KUKA KRL program: MyProgram_034().src

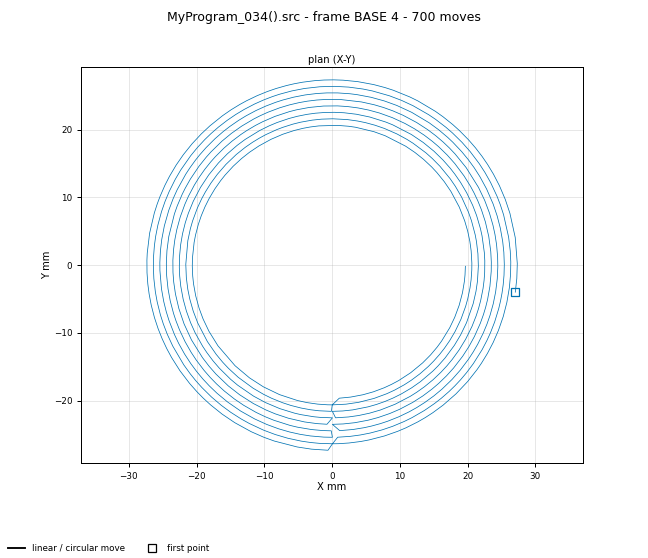
[picture p0: tool path of MyProgram_034().src in frame BASE 4, 700 of 700 moves have a stored position in this frame; points joined in program order, loops and branches not executed]
&ACCESS RVP
&REL 1
&PARAM TEMPLATE = C:\KRC\Roboter\Template\vorgabe
&PARAM EDITMASK = *
DEF MyProgram_034()
; ---- Setting reference (Base) ----
$BASE = BASE_DATA[4]

; --------------------------
; ---- Setting tool (TCP) ----
$TOOL = TOOL_DATA[3]
; --------------------------

$VEL.CP = VEL_APROX_PRINT
Startdeposition()
$VEL.CP = VEL_PRINT
LIN {X 27.0548,Y -4.0022,Z 60,A -14.7192,B 24.8252,C -3.0498,E1 25.1584,E2 -622.5769} C_DIS
LIN {X 27.276,Y -1.9895,Z 60,A -9.9625,B 24.8229,C -3.0695,E1 25.1596,E2 -627.352} C_DIS
LIN {X 27.3471,Y 0.2163,Z 60,A -4.9436,B 24.8206,C -3.0888,E1 25.1596,E2 -632.3869} C_DIS
LIN {X 27.0427,Y 4.0823,Z 60,A 3.1933,B 24.8177,C -3.1139,E1 25.1571,E2 -640.5351} C_DIS
LIN {X 26.2619,Y 7.6301,Z 60,A 9.5753,B 24.8168,C -3.1215,E1 25.1528,E2 -646.8981} C_DIS
LIN {X 25.5723,Y 9.6957,Z 60,A 14.6425,B 24.8145,C -3.1407,E1 25.1481,E2 -651.9824} C_DIS
LIN {X 24.7146,Y 11.7115,Z 60,A 18.9352,B 24.8135,C -3.1497,E1 25.1432,E2 -656.2733} C_DIS
LIN {X 23.8276,Y 13.424,Z 60,A 22.7576,B 24.8125,C -3.1579,E1 25.1381,E2 -660.0948} C_DIS
LIN {X 22.9582,Y 14.8622,Z 60,A 26.1439,B 24.8116,C -3.1652,E1 25.1331,E2 -663.4815} C_DIS
LIN {X 22.1384,Y 16.0578,Z 60,A 28.9814,B 24.811,C -3.1703,E1 25.1285,E2 -666.3172} C_DIS
LIN {X 21.1745,Y 17.3093,Z 60,A 32.8226,B 24.8093,C -3.1841,E1 25.1218,E2 -670.1731} C_DIS
LIN {X 20.1397,Y 18.5025,Z 60,A 35.9451,B 24.8087,C -3.1892,E1 25.116,E2 -673.2939} C_DIS
LIN {X 18.8106,Y 19.8529,Z 60,A 39.9521,B 24.8077,C -3.1977,E1 25.108,E2 -677.3042} C_DIS
LIN {X 17.8285,Y 20.7391,Z 60,A 42.6684,B 24.8071,C -3.2024,E1 25.1023,E2 -680.0209} C_DIS
LIN {X 16.3808,Y 21.9002,Z 60,A 46.4204,B 24.8065,C -3.2077,E1 25.094,E2 -683.7718} C_DIS
LIN {X 15.2507,Y 22.7016,Z 60,A 50.0968,B 24.8049,C -3.2207,E1 25.0855,E2 -687.4666} C_DIS
LIN {X 12.664,Y 24.2399,Z 60,A 55.4757,B 24.8051,C -3.2195,E1 25.0725,E2 -692.8267} C_DIS
LIN {X 11.4734,Y 24.8254,Z 60,A 58.7236,B 24.8041,C -3.2275,E1 25.0642,E2 -696.0853} C_DIS
LIN {X 9.042,Y 25.8106,Z 60,A 63.8728,B 24.8039,C -3.2292,E1 25.0508,E2 -701.2272} C_DIS
LIN {X 7.8177,Y 26.2072,Z 60,A 66.6148,B 24.8036,C -3.2316,E1 25.0435,E2 -703.97} C_DIS
LIN {X 6.141,Y 26.6504,Z 60,A 70.1776,B 24.8034,C -3.2329,E1 25.0339,E2 -707.5308} C_DIS
LIN {X 3.7878,Y 27.0854,Z 60,A 75.9719,B 24.8023,C -3.2419,E1 25.0179,E2 -713.3405} C_DIS
LIN {X 1.6343,Y 27.2996,Z 60,A 79.5933,B 24.8033,C -3.2337,E1 25.0078,E2 -716.9407} C_DIS
LIN {X 0.2341,Y 27.348,Z 60,A 82.5895,B 24.8033,C -3.2339,E1 24.9995,E2 -719.9368} C_DIS
LIN {X -1.1756,Y 27.3235,Z 60,A 85.9478,B 24.803,C -3.2366,E1 24.9901,E2 -723.3021} C_DIS
LIN {X -2.5854,Y 27.2262,Z 60,A 88.7053,B 24.8034,C -3.2334,E1 24.9824,E2 -726.0534} C_DIS
LIN {X -4.3352,Y 27.003,Z 60,A 92.0727,B 24.804,C -3.2283,E1 24.9731,E2 -729.4114} C_DIS
LIN {X -5.5747,Y 26.7748,Z 60,A 94.7372,B 24.8042,C -3.2265,E1 24.9658,E2 -732.0744} C_DIS
LIN {X -6.7187,Y 26.5103,Z 60,A 97.2104,B 24.8045,C -3.2243,E1 24.9591,E2 -734.5458} C_DIS
LIN {X -8.2695,Y 26.0682,Z 60,A 100.3423,B 24.8051,C -3.2187,E1 24.9508,E2 -737.6697} C_DIS
LIN {X -9.553,Y 25.6257,Z 60,A 103.726,B 24.8051,C -3.2195,E1 24.9419,E2 -741.0618} C_DIS
LIN {X -11.0562,Y 25.0141,Z 60,A 107.0784,B 24.8057,C -3.2144,E1 24.9333,E2 -744.4097} C_DIS
LIN {X -12.6311,Y 24.2572,Z 60,A 110.2156,B 24.8068,C -3.2047,E1 24.9254,E2 -747.5321} C_DIS
LIN {X -13.6382,Y 23.7057,Z 60,A 112.807,B 24.8072,C -3.2021,E1 24.9191,E2 -750.1246} C_DIS
LIN {X -14.9175,Y 22.9225,Z 60,A 116.3286,B 24.8075,C -3.1991,E1 24.9108,E2 -753.6502} C_DIS
LIN {X -16.1878,Y 22.0436,Z 60,A 119.8069,B 24.8081,C -3.1944,E1 24.9029,E2 -757.1295} C_DIS
LIN {X -18.0508,Y 20.546,Z 60,A 124.7797,B 24.8094,C -3.1834,E1 24.8923,E2 -762.0951} C_DIS
LIN {X -19.3253,Y 19.3515,Z 60,A 128.3639,B 24.8105,C -3.1744,E1 24.8851,E2 -765.6727} C_DIS
LIN {X -20.6728,Y 17.905,Z 60,A 133.0331,B 24.8113,C -3.1678,E1 24.8764,E2 -770.347} C_DIS
LIN {X -21.9574,Y 16.304,Z 60,A 136.9144,B 24.813,C -3.1539,E1 24.8698,E2 -774.2135} C_DIS
LIN {X -23.0224,Y 14.7624,Z 60,A 140.9378,B 24.8141,C -3.1439,E1 24.8636,E2 -778.2331} C_DIS
LIN {X -24.0135,Y 13.0887,Z 60,A 144.7588,B 24.8157,C -3.1309,E1 24.8583,E2 -782.0428} C_DIS
LIN {X -24.6915,Y 11.7597,Z 60,A 148.0146,B 24.8167,C -3.1227,E1 24.8543,E2 -785.2965} C_DIS
LIN {X -25.4087,Y 10.1165,Z 60,A 151.5582,B 24.8181,C -3.1103,E1 24.8505,E2 -788.8302} C_DIS
LIN {X -25.8191,Y 9.0175,Z 60,A 154.1643,B 24.8189,C -3.1038,E1 24.8481,E2 -791.4355} C_DIS
LIN {X -26.2429,Y 7.6978,Z 60,A 157.7395,B 24.8194,C -3.0991,E1 24.8452,E2 -795.02} C_DIS
LIN {X -26.9423,Y 4.7003,Z 60,A 164.4262,B 24.8216,C -3.0806,E1 24.8414,E2 -801.7017} C_DIS
LIN {X -27.2903,Y 1.7841,Z 60,A 169.5574,B 24.8245,C -3.0552,E1 24.84,E2 -806.8029} C_DIS
LIN {X -27.3397,Y 0.7102,Z 60,A 172.2916,B 24.825,C -3.0511,E1 24.8398,E2 -809.5437} C_DIS
LIN {X -27.3254,Y -1.1279,Z 60,A 176.1128,B 24.8264,C -3.0389,E1 24.84,E2 -813.3588} C_DIS
LIN {X -27.2072,Y -2.7805,Z 60,A 179.4041,B 24.8278,C -3.0271,E1 24.8408,E2 -816.6416} C_DIS
LIN {X -27.0158,Y -4.2561,Z 60,A -177.359,B 24.8288,C -3.0183,E1 24.8421,E2 -819.8767} C_DIS
LIN {X -26.7044,Y -5.9026,Z 60,A -173.7332,B 24.8299,C -3.0085,E1 24.8442,E2 -823.5003} C_DIS
LIN {X -26.2251,Y -7.7583,Z 60,A -169.3981,B 24.831,C -2.9986,E1 24.8474,E2 -827.837} C_DIS
LIN {X -25.681,Y -9.4042,Z 60,A -166.0791,B 24.8324,C -2.9862,E1 24.8505,E2 -831.1452} C_DIS
LIN {X -25.091,Y -10.8804,Z 60,A -163.0196,B 24.8336,C -2.9752,E1 24.8538,E2 -834.1952} C_DIS
LIN {X -24.4098,Y -12.3345,Z 60,A -159.3572,B 24.8344,C -2.968,E1 24.8582,E2 -837.8602} C_DIS
LIN {X -23.7002,Y -13.6473,Z 60,A -156.0691,B 24.8352,C -2.9609,E1 24.8627,E2 -841.1485} C_DIS
LIN {X -22.4555,Y -15.6113,Z 60,A -150.8,B 24.8363,C -2.9515,E1 24.8709,E2 -846.4215} C_DIS
LIN {X -21.0274,Y -17.4874,Z 60,A -146.2708,B 24.8379,C -2.9373,E1 24.8787,E2 -850.938} C_DIS
LIN {X -19.9376,Y -18.7205,Z 60,A -143.0013,B 24.8388,C -2.9286,E1 24.8848,E2 -854.2012} C_DIS
LIN {X -19.0275,Y -19.6448,Z 60,A -140.3601,B 24.8395,C -2.9225,E1 24.8901,E2 -856.839} C_DIS
LIN {X -17.962,Y -20.6236,Z 60,A -137.0049,B 24.8399,C -2.9191,E1 24.8971,E2 -860.1993} C_DIS
LIN {X -16.2373,Y -22.0074,Z 60,A -131.962,B 24.8404,C -2.9142,E1 24.9083,E2 -865.2488} C_DIS
LIN {X -14.3669,Y -23.2712,Z 60,A -127.2621,B 24.8412,C -2.9069,E1 24.9193,E2 -869.9464} C_DIS
LIN {X -11.9291,Y -24.6102,Z 60,A -121.5891,B 24.8422,C -2.8984,E1 24.9333,E2 -875.6147} C_DIS
LIN {X -10.075,Y -25.4254,Z 60,A -117.4657,B 24.8427,C -2.8932,E1 24.9439,E2 -879.735} C_DIS
LIN {X -8.5417,Y -25.9801,Z 60,A -113.2565,B 24.8423,C -2.8973,E1 24.9551,E2 -883.9619} C_DIS
LIN {X -5.1473,Y -26.86,Z 60,A -107.1176,B 24.8438,C -2.883,E1 24.9717,E2 -890.075} C_DIS
LIN {X -3.0426,Y -27.1795,Z 60,A -101.5966,B 24.8429,C -2.8918,E1 24.9871,E2 -895.6211} C_DIS
LIN {X -0.6027,Y -27.3425,Z 60,A -97.5116,B 24.8439,C -2.8825,E1 24.9984,E2 -899.6849} C_DIS
LIN {X -0.6027,Y -27.3425,Z 60,A -97.5116,B 24.8439,C -2.8825,E1 24.9984,E2 -899.6849} C_DIS
Enddeposition()
LIN {X 0.0589,Y -26.3872,Z 60,A -97.338,B 24.8433,C -2.8883,E1 24.9989,E2 -899.8724} C_DIS
Startdeposition()
$VEL.CP = VEL_PRINT
LIN {X -1.8545,Y -26.3253,Z 60,A -101.7289,B 24.8435,C -2.8859,E1 24.9867,E2 -895.4746} C_DIS
LIN {X -3.1824,Y -26.198,Z 60,A -104.3677,B 24.8432,C -2.8884,E1 24.9794,E2 -892.8403} C_DIS
LIN {X -4.5794,Y -25.9906,Z 60,A -107.6972,B 24.8434,C -2.887,E1 24.9702,E2 -889.5044} C_DIS
LIN {X -6.5439,Y -25.5663,Z 60,A -112.5834,B 24.8436,C -2.8849,E1 24.9569,E2 -884.6068} C_DIS
LIN {X -8.376,Y -25.0259,Z 60,A -116.0454,B 24.8427,C -2.8933,E1 24.9477,E2 -881.1587} C_DIS
LIN {X -10.101,Y -24.3809,Z 60,A -120.796,B 24.8429,C -2.8913,E1 24.9353,E2 -876.3929} C_DIS
LIN {X -12.22,Y -23.3909,Z 60,A -125.0898,B 24.8416,C -2.9031,E1 24.9246,E2 -872.116} C_DIS
LIN {X -13.4081,Y -22.731,Z 60,A -128.3851,B 24.8415,C -2.9046,E1 24.9166,E2 -868.8145} C_DIS
LIN {X -14.9597,Y -21.7411,Z 60,A -131.9408,B 24.8405,C -2.9138,E1 24.9083,E2 -865.2692} C_DIS
LIN {X -16.352,Y -20.7143,Z 60,A -136.4907,B 24.8404,C -2.9147,E1 24.8982,E2 -860.7052} C_DIS
LIN {X -17.8054,Y -19.4789,Z 60,A -140.2956,B 24.8392,C -2.9249,E1 24.8902,E2 -856.9093} C_DIS
LIN {X -19.2341,Y -18.0698,Z 60,A -144.562,B 24.8382,C -2.9344,E1 24.8819,E2 -852.6477} C_DIS
LIN {X -20.1352,Y -17.0603,Z 60,A -147.365,B 24.8374,C -2.9418,E1 24.8767,E2 -849.8496} C_DIS
LIN {X -20.9498,Y -16.0494,Z 60,A -150.3147,B 24.8367,C -2.9475,E1 24.8717,E2 -846.8996} C_DIS
LIN {X -21.8937,Y -14.7357,Z 60,A -154.7545,B 24.8364,C -2.9504,E1 24.8646,E2 -842.4449} C_DIS
LIN {X -23.5206,Y -11.969,Z 60,A -160.9111,B 24.8338,C -2.9735,E1 24.8563,E2 -836.3111} C_DIS
LIN {X -24.3328,Y -10.2164,Z 60,A -165.4742,B 24.8328,C -2.9829,E1 24.8511,E2 -831.7455} C_DIS
LIN {X -24.9188,Y -8.6894,Z 60,A -168.4952,B 24.8313,C -2.9961,E1 24.8482,E2 -828.739} C_DIS
LIN {X -25.3556,Y -7.3183,Z 60,A -171.8754,B 24.8304,C -3.0038,E1 24.8455,E2 -825.3577} C_DIS
LIN {X -25.8217,Y -5.4498,Z 60,A -176.6121,B 24.8293,C -3.0132,E1 24.8425,E2 -820.6158} C_DIS
LIN {X -26.0936,Y -3.9506,Z 60,A -179.4841,B 24.8279,C -3.0256,E1 24.8412,E2 -817.7565} C_DIS
LIN {X -26.3148,Y -1.9967,Z 60,A 176.035,B 24.8266,C -3.0376,E1 24.84,E2 -813.2775} C_DIS
LIN {X -26.3891,Y -0.2353,Z 60,A 172.4842,B 24.825,C -3.051,E1 24.8398,E2 -809.7374} C_DIS
LIN {X -26.3608,Y 1.251,Z 60,A 169.2644,B 24.8238,C -3.0611,E1 24.8401,E2 -806.5224} C_DIS
LIN {X -26.2322,Y 2.8893,Z 60,A 165.3007,B 24.8228,C -3.0701,E1 24.8411,E2 -802.5565} C_DIS
LIN {X -26.0485,Y 4.2383,Z 60,A 162.277,B 24.8218,C -3.079,E1 24.8424,E2 -799.5359} C_DIS
LIN {X -25.721,Y 5.9053,Z 60,A 158.6703,B 24.8204,C -3.0908,E1 24.8445,E2 -795.9363} C_DIS
LIN {X -25.1844,Y 7.8876,Z 60,A 154.2854,B 24.8188,C -3.1048,E1 24.8479,E2 -791.5596} C_DIS
LIN {X -24.6568,Y 9.4086,Z 60,A 150.9955,B 24.8174,C -3.1164,E1 24.8511,E2 -788.2788} C_DIS
LIN {X -24.0603,Y 10.8427,Z 60,A 147.5968,B 24.8162,C -3.1262,E1 24.8548,E2 -784.8847} C_DIS
LIN {X -23.1656,Y 12.6425,Z 60,A 142.4262,B 24.8153,C -3.1341,E1 24.8615,E2 -779.7055} C_DIS
LIN {X -22.3606,Y 14.017,Z 60,A 138.9318,B 24.8142,C -3.1434,E1 24.8666,E2 -776.2156} C_DIS
LIN {X -20.876,Y 16.1453,Z 60,A 134.1223,B 24.8119,C -3.163,E1 24.8745,E2 -771.4298} C_DIS
LIN {X -19.8722,Y 17.3657,Z 60,A 130.357,B 24.8111,C -3.1696,E1 24.8813,E2 -767.6631} C_DIS
LIN {X -18.8133,Y 18.5077,Z 60,A 127.158,B 24.81,C -3.1788,E1 24.8874,E2 -764.4722} C_DIS
LIN {X -17.8869,Y 19.4046,Z 60,A 124.5015,B 24.8091,C -3.1861,E1 24.8928,E2 -761.8222} C_DIS
LIN {X -16.7757,Y 20.3731,Z 60,A 120.7979,B 24.8087,C -3.1898,E1 24.9007,E2 -758.1132} C_DIS
LIN {X -15.4967,Y 21.3619,Z 60,A 117.8887,B 24.8073,C -3.2008,E1 24.9072,E2 -755.2199} C_DIS
LIN {X -14.2447,Y 22.2163,Z 60,A 113.9784,B 24.8071,C -3.2029,E1 24.9163,E2 -751.3016} C_DIS
LIN {X -12.9681,Y 22.9848,Z 60,A 110.842,B 24.8063,C -3.2091,E1 24.9239,E2 -748.1709} C_DIS
LIN {X -11.4385,Y 23.7829,Z 60,A 107.0049,B 24.8057,C -3.2144,E1 24.9334,E2 -744.3361} C_DIS
LIN {X -10.0968,Y 24.3829,Z 60,A 104.1164,B 24.8049,C -3.221,E1 24.9408,E2 -741.4567} C_DIS
LIN {X -8.8017,Y 24.879,Z 60,A 101.2584,B 24.8043,C -3.2259,E1 24.9483,E2 -738.6046} C_DIS
LIN {X -7.7742,Y 25.2194,Z 60,A 98.5223,B 24.8043,C -3.2257,E1 24.9556,E2 -735.8631} C_DIS
LIN {X -5.9465,Y 25.712,Z 60,A 94.8843,B 24.8034,C -3.2332,E1 24.9654,E2 -732.2378} C_DIS
LIN {X -4.073,Y 26.0746,Z 60,A 89.7625,B 24.8039,C -3.2286,E1 24.9795,E2 -727.0999} C_DIS
LIN {X -1.7766,Y 26.3308,Z 60,A 85.1531,B 24.8033,C -3.2343,E1 24.9923,E2 -722.5016} C_DIS
LIN {X 0.3913,Y 26.3881,Z 60,A 80.1495,B 24.8034,C -3.2328,E1 25.0063,E2 -717.4946} C_DIS
LIN {X 2.4435,Y 26.2772,Z 60,A 75.8887,B 24.8032,C -3.2344,E1 25.0181,E2 -713.2395} C_DIS
LIN {X 4.5446,Y 25.9965,Z 60,A 71.6018,B 24.8031,C -3.2359,E1 25.03,E2 -708.9602} C_DIS
LIN {X 5.9537,Y 25.7103,Z 60,A 67.9541,B 24.8038,C -3.2296,E1 25.0399,E2 -705.3025} C_DIS
LIN {X 8.4767,Y 24.9923,Z 60,A 62.7874,B 24.8038,C -3.2304,E1 25.0537,E2 -700.1468} C_DIS
LIN {X 10.245,Y 24.3208,Z 60,A 58.2968,B 24.8047,C -3.2227,E1 25.0654,E2 -695.6482} C_DIS
LIN {X 11.9465,Y 23.5321,Z 60,A 53.9882,B 24.8055,C -3.2156,E1 25.0762,E2 -691.334} C_DIS
LIN {X 14.2708,Y 22.1988,Z 60,A 49.2529,B 24.8052,C -3.2181,E1 25.0875,E2 -686.6192} C_DIS
LIN {X 15.2838,Y 21.5147,Z 60,A 45.7841,B 24.8068,C -3.2055,E1 25.0955,E2 -683.1324} C_DIS
LIN {X 16.7912,Y 20.3598,Z 60,A 42.2398,B 24.8069,C -3.2041,E1 25.1032,E2 -679.5981} C_DIS
LIN {X 17.7707,Y 19.5111,Z 60,A 39.2592,B 24.8078,C -3.1969,E1 25.1094,E2 -676.6123} C_DIS
LIN {X 19.1933,Y 18.1134,Z 60,A 34.2905,B 24.8097,C -3.1811,E1 25.1192,E2 -671.6274} C_DIS
LIN {X 20.3945,Y 16.7497,Z 60,A 30.593,B 24.8104,C -3.1749,E1 25.1258,E2 -667.9319} C_DIS
LIN {X 21.7332,Y 14.9711,Z 60,A 26.0293,B 24.8115,C -3.1662,E1 25.1333,E2 -663.3698} C_DIS
LIN {X 22.5669,Y 13.6825,Z 60,A 23.185,B 24.8118,C -3.1632,E1 25.1375,E2 -660.5327} C_DIS
LIN {X 23.4068,Y 12.1896,Z 60,A 18.6048,B 24.8142,C -3.1437,E1 25.1436,E2 -655.9303} C_DIS
LIN {X 24.357,Y 10.1587,Z 60,A 14.6173,B 24.8146,C -3.1402,E1 25.1481,E2 -651.9563} C_DIS
LIN {X 24.8411,Y 8.9095,Z 60,A 11.3299,B 24.8161,C -3.1276,E1 25.1513,E2 -648.6573} C_DIS
LIN {X 25.3233,Y 7.4287,Z 60,A 7.148,B 24.8183,C -3.1085,E1 25.1547,E2 -644.454} C_DIS
LIN {X 26.066,Y 4.1287,Z 60,A 0.809,B 24.8196,C -3.098,E1 25.1582,E2 -638.1271} C_DIS
LIN {X 26.3079,Y 2.087,Z 60,A -4.1531,B 24.8218,C -3.0784,E1 25.1595,E2 -633.148} C_DIS
LIN {X 26.3868,Y 0.4595,Z 60,A -7.2624,B 24.8225,C -3.0724,E1 25.1598,E2 -630.0429} C_DIS
LIN {X 26.3574,Y -1.3178,Z 60,A -11.2637,B 24.8241,C -3.0587,E1 25.1594,E2 -626.033} C_DIS
LIN {X 26.1796,Y -3.3321,Z 60,A -15.5934,B 24.8256,C -3.0456,E1 25.1581,E2 -621.698} C_DIS
LIN {X 25.8041,Y -5.5322,Z 60,A -20.1106,B 24.8269,C -3.0345,E1 25.1558,E2 -617.1807} C_DIS
LIN {X 25.2681,Y -7.613,Z 60,A -25.1505,B 24.8291,C -3.0158,E1 25.152,E2 -612.1255} C_DIS
LIN {X 24.5603,Y -9.6565,Z 60,A -29.8268,B 24.8306,C -3.0019,E1 25.1475,E2 -607.4425} C_DIS
LIN {X 23.7829,Y -11.4385,Z 60,A -33.916,B 24.8319,C -2.9911,E1 25.1427,E2 -603.3498} C_DIS
LIN {X 22.9344,Y -13.0576,Z 60,A -37.6543,B 24.8328,C -2.9824,E1 25.1377,E2 -599.6105} C_DIS
LIN {X 22.0532,Y -14.4954,Z 60,A -40.7767,B 24.8333,C -2.9785,E1 25.133,E2 -596.4946} C_DIS
LIN {X 21.4128,Y -15.4265,Z 60,A -44.2639,B 24.8353,C -2.9602,E1 25.1274,E2 -592.981} C_DIS
LIN {X 20.0147,Y -17.2014,Z 60,A -48.9008,B 24.8364,C -2.9507,E1 25.1191,E2 -588.343} C_DIS
LIN {X 18.3038,Y -19.0117,Z 60,A -54.5985,B 24.8382,C -2.9347,E1 25.1079,E2 -582.6315} C_DIS
LIN {X 16.3947,Y -20.6805,Z 60,A -59.499,B 24.8388,C -2.9293,E1 25.0974,E2 -577.7369} C_DIS
LIN {X 14.8639,Y -21.8067,Z 60,A -62.9575,B 24.8388,C -2.9281,E1 25.0896,E2 -574.2879} C_DIS
LIN {X 13.7669,Y -22.5155,Z 60,A -66.1412,B 24.8399,C -2.9191,E1 25.0821,E2 -571.0932} C_DIS
LIN {X 12.6901,Y -23.1396,Z 60,A -69.2111,B 24.8408,C -2.9107,E1 25.0745,E2 -568.0122} C_DIS
LIN {X 10.8993,Y -24.0349,Z 60,A -73.3326,B 24.8413,C -2.9062,E1 25.0642,E2 -563.8909} C_DIS
LIN {X 9.6687,Y -24.5557,Z 60,A -76.598,B 24.8421,C -2.8986,E1 25.0557,E2 -560.6147} C_DIS
LIN {X 7.7271,Y -25.2339,Z 60,A -81.0311,B 24.8427,C -2.8936,E1 25.0439,E2 -556.1783} C_DIS
LIN {X 5.4433,Y -25.8233,Z 60,A -85.2517,B 24.8423,C -2.8974,E1 25.0325,E2 -551.9727} C_DIS
LIN {X 4.2391,Y -26.0483,Z 60,A -88.6171,B 24.8432,C -2.8886,E1 25.0232,E2 -548.5902} C_DIS
LIN {X 2.4827,Y -26.2735,Z 60,A -92.2516,B 24.8432,C -2.8884,E1 25.0131,E2 -544.9577} C_DIS
LIN {X 0.9605,Y -26.3727,Z 60,A -95.4196,B 24.8432,C -2.8884,E1 25.0043,E2 -541.7908} C_DIS
LIN {X 0.0589,Y -26.3872,Z 60,A -97.3379,B 24.8432,C -2.8883,E1 24.9989,E2 -539.8724} C_DIS
Enddeposition()
LIN {X 0.0589,Y -26.3872,Z 60,A -97.3379,B 24.8432,C -2.8883,E1 24.9989,E2 -539.8724} C_DIS
Startdeposition()
$VEL.CP = VEL_PRINT
LIN {X 0.8302,Y -25.4191,Z 60,A -93.7064,B 24.8395,C -2.9222,E1 25.0093,E2 -543.584} C_DIS
LIN {X 2.6635,Y -25.2926,Z 60,A -90.047,B 24.8398,C -2.9199,E1 25.0195,E2 -547.2359} C_DIS
LIN {X 4.159,Y -25.0903,Z 60,A -86.6827,B 24.8396,C -2.9219,E1 25.0288,E2 -550.6019} C_DIS
LIN {X 5.6318,Y -24.801,Z 60,A -83.0518,B 24.839,C -2.9273,E1 25.0387,E2 -554.2407} C_DIS
LIN {X 7.4181,Y -24.3265,Z 60,A -79.1443,B 24.8388,C -2.9292,E1 25.0492,E2 -558.1464} C_DIS
LIN {X 8.9447,Y -23.8073,Z 60,A -75.4107,B 24.8381,C -2.9348,E1 25.059,E2 -561.8857} C_DIS
LIN {X 10.6425,Y -23.0984,Z 60,A -71.3614,B 24.8376,C -2.9399,E1 25.0694,E2 -565.9372} C_DIS
LIN {X 11.8063,Y -22.5259,Z 60,A -68.0719,B 24.8366,C -2.9485,E1 25.0776,E2 -569.2378} C_DIS
LIN {X 13.6252,Y -21.4752,Z 60,A -63.6418,B 24.836,C -2.9538,E1 25.0881,E2 -573.667} C_DIS
LIN {X 15.1129,Y -20.4555,Z 60,A -59.7145,B 24.8353,C -2.9605,E1 25.0971,E2 -577.5964} C_DIS
LIN {X 16.1132,Y -19.6774,Z 60,A -57.1199,B 24.8349,C -2.9638,E1 25.1027,E2 -580.189} C_DIS
LIN {X 17.2639,Y -18.6756,Z 60,A -53.7628,B 24.8342,C -2.9706,E1 25.1098,E2 -583.5489} C_DIS
LIN {X 18.1315,Y -17.8344,Z 60,A -50.8373,B 24.8332,C -2.9792,E1 25.1156,E2 -586.4826} C_DIS
LIN {X 18.9507,Y -16.9615,Z 60,A -47.8025,B 24.832,C -2.9896,E1 25.1213,E2 -589.5286} C_DIS
LIN {X 19.8632,Y -15.8827,Z 60,A -44.764,B 24.8313,C -2.9962,E1 25.1267,E2 -592.5685} C_DIS
LIN {X 20.8593,Y -14.5503,Z 60,A -40.8226,B 24.8299,C -3.0083,E1 25.1331,E2 -596.5196} C_DIS
LIN {X 22.1504,Y -12.4978,Z 60,A -35.5632,B 24.8284,C -3.0212,E1 25.1407,E2 -601.7827} C_DIS
LIN {X 22.863,Y -11.1399,Z 60,A -32.4452,B 24.8277,C -3.0273,E1 25.1446,E2 -604.8986} C_DIS
LIN {X 23.3731,Y -10.0244,Z 60,A -29.4266,B 24.8265,C -3.0384,E1 25.148,E2 -607.927} C_DIS
LIN {X 24.0018,Y -8.4094,Z 60,A -25.4521,B 24.825,C -3.051,E1 25.1518,E2 -611.909} C_DIS
LIN {X 24.5997,Y -6.4544,Z 60,A -21.2805,B 24.824,C -3.06,E1 25.155,E2 -616.0781} C_DIS
LIN {X 24.876,Y -5.2908,Z 60,A -18.673,B 24.8231,C -3.0673,E1 25.1566,E2 -618.6878} C_DIS
LIN {X 25.0946,Y -4.1333,Z 60,A -15.9329,B 24.8221,C -3.0766,E1 25.158,E2 -621.4337} C_DIS
LIN {X 25.2651,Y -2.9136,Z 60,A -13.2149,B 24.8211,C -3.0846,E1 25.1589,E2 -624.1547} C_DIS
LIN {X 25.3889,Y -1.4849,Z 60,A -9.7203,B 24.8196,C -3.0978,E1 25.1596,E2 -627.6598} C_DIS
LIN {X 25.431,Y 0.091,Z 60,A -6.2312,B 24.8184,C -3.1082,E1 25.1597,E2 -631.1527} C_DIS
LIN {X 25.3626,Y 1.8812,Z 60,A -2.4671,B 24.8173,C -3.1175,E1 25.1592,E2 -634.9165} C_DIS
LIN {X 25.1924,Y 3.4867,Z 60,A 1.3741,B 24.8157,C -3.131,E1 25.1579,E2 -638.7672} C_DIS
LIN {X 24.8385,Y 5.4646,Z 60,A 6.3509,B 24.8134,C -3.1499,E1 25.1552,E2 -643.7596} C_DIS
LIN {X 24.3699,Y 7.2747,Z 60,A 9.8564,B 24.8129,C -3.1542,E1 25.1525,E2 -647.2551} C_DIS
LIN {X 23.779,Y 9.0204,Z 60,A 14.9051,B 24.8103,C -3.1763,E1 25.1477,E2 -652.3281} C_DIS
LIN {X 22.8138,Y 11.2393,Z 60,A 19.7864,B 24.8093,C -3.1848,E1 25.142,E2 -657.2031} C_DIS
LIN {X 21.8294,Y 13.0503,Z 60,A 24.4006,B 24.8078,C -3.1966,E1 25.1356,E2 -661.8212} C_DIS
LIN {X 20.9749,Y 14.3831,Z 60,A 27.4988,B 24.8074,C -3.2003,E1 25.1308,E2 -664.9129} C_DIS
LIN {X 20.1222,Y 15.5536,Z 60,A 31.1996,B 24.8059,C -3.2128,E1 25.1246,E2 -668.6257} C_DIS
LIN {X 19.1468,Y 16.7398,Z 60,A 34.6365,B 24.805,C -3.2203,E1 25.1183,E2 -672.0647} C_DIS
LIN {X 17.8273,Y 18.1385,Z 60,A 38.412,B 24.8046,C -3.2234,E1 25.111,E2 -675.8315} C_DIS
LIN {X 17.0875,Y 18.8372,Z 60,A 41.0209,B 24.8036,C -3.2313,E1 25.1056,E2 -678.4484} C_DIS
LIN {X 15.7412,Y 19.9759,Z 60,A 45.2287,B 24.8024,C -3.2409,E1 25.0965,E2 -682.6632} C_DIS
LIN {X 14.3367,Y 21.0068,Z 60,A 49.5827,B 24.8011,C -3.2516,E1 25.0865,E2 -687.0276} C_DIS
LIN {X 11.7479,Y 22.5558,Z 60,A 55.8392,B 24.8006,C -3.2555,E1 25.0713,E2 -693.2748} C_DIS
LIN {X 9.5413,Y 23.5745,Z 60,A 61.5013,B 24.7997,C -3.2632,E1 25.0568,E2 -698.9413} C_DIS
LIN {X 7.7095,Y 24.2355,Z 60,A 65.8073,B 24.7994,C -3.2659,E1 25.0455,E2 -703.2456} C_DIS
LIN {X 5.7665,Y 24.7703,Z 60,A 70.2897,B 24.7991,C -3.268,E1 25.0333,E2 -707.7263} C_DIS
LIN {X 3.6985,Y 25.1618,Z 60,A 74.4174,B 24.7996,C -3.2643,E1 25.022,E2 -711.8406} C_DIS
LIN {X 2.6271,Y 25.2965,Z 60,A 77.4616,B 24.7989,C -3.2699,E1 25.0135,E2 -714.8961} C_DIS
LIN {X 0.8212,Y 25.4194,Z 60,A 81.2445,B 24.7992,C -3.2672,E1 25.003,E2 -718.6713} C_DIS
LIN {X -0.7596,Y 25.4212,Z 60,A 84.922,B 24.7992,C -3.2673,E1 24.9927,E2 -722.3494} C_DIS
LIN {X -2.2712,Y 25.3311,Z 60,A 88.1256,B 24.7996,C -3.2642,E1 24.9838,E2 -725.5468} C_DIS
LIN {X -3.9675,Y 25.1214,Z 60,A 92.5631,B 24.7993,C -3.2664,E1 24.9715,E2 -729.9931} C_DIS
LIN {X -5.6558,Y 24.7957,Z 60,A 95.8732,B 24.8002,C -3.2589,E1 24.9625,E2 -733.2892} C_DIS
LIN {X -7.2639,Y 24.3731,Z 60,A 99.3157,B 24.801,C -3.2529,E1 24.9533,E2 -736.7227} C_DIS
LIN {X -8.3177,Y 24.0338,Z 60,A 102.228,B 24.801,C -3.2529,E1 24.9456,E2 -739.6406} C_DIS
LIN {X -9.7872,Y 23.4738,Z 60,A 105.9363,B 24.8014,C -3.2494,E1 24.936,E2 -743.3486} C_DIS
LIN {X -11.2454,Y 22.811,Z 60,A 109.6677,B 24.802,C -3.2448,E1 24.9266,E2 -747.0785} C_DIS
LIN {X -12.6998,Y 22.0349,Z 60,A 113.043,B 24.803,C -3.2362,E1 24.9183,E2 -750.4431} C_DIS
LIN {X -13.8147,Y 21.3534,Z 60,A 115.8771,B 24.8038,C -3.2302,E1 24.9117,E2 -753.2717} C_DIS
LIN {X -15.1237,Y 20.4477,Z 60,A 119.275,B 24.8048,C -3.2219,E1 24.9039,E2 -756.6615} C_DIS
LIN {X -16.1076,Y 19.6819,Z 60,A 122.6671,B 24.805,C -3.2197,E1 24.8965,E2 -760.0611} C_DIS
LIN {X -17.2919,Y 18.6494,Z 60,A 126.2739,B 24.8059,C -3.2123,E1 24.8891,E2 -763.6644} C_DIS
LIN {X -18.5881,Y 17.358,Z 60,A 130.1453,B 24.8073,C -3.201,E1 24.8815,E2 -767.5254} C_DIS
LIN {X -19.5433,Y 16.2751,Z 60,A 133.1897,B 24.8084,C -3.1916,E1 24.876,E2 -770.5613} C_DIS
LIN {X -20.1888,Y 15.4673,Z 60,A 135.7592,B 24.809,C -3.187,E1 24.8716,E2 -773.132} C_DIS
LIN {X -20.9954,Y 14.353,Z 60,A 138.7404,B 24.8101,C -3.1781,E1 24.8668,E2 -776.1065} C_DIS
LIN {X -21.6141,Y 13.4037,Z 60,A 141.9783,B 24.8104,C -3.175,E1 24.862,E2 -779.3535} C_DIS
LIN {X -22.8705,Y 11.1248,Z 60,A 147.4345,B 24.8127,C -3.156,E1 24.8549,E2 -784.7932} C_DIS
LIN {X -23.4723,Y 9.7908,Z 60,A 150.9419,B 24.8137,C -3.1475,E1 24.851,E2 -788.2995} C_DIS
LIN {X -24.1147,Y 8.0795,Z 60,A 155.0695,B 24.8152,C -3.1352,E1 24.8472,E2 -792.4211} C_DIS
LIN {X -24.7652,Y 5.788,Z 60,A 161.0217,B 24.8167,C -3.1219,E1 24.843,E2 -798.3761} C_DIS
LIN {X -25.1517,Y 3.7705,Z 60,A 164.9807,B 24.8189,C -3.104,E1 24.8412,E2 -802.3156} C_DIS
LIN {X -25.3452,Y 2.1031,Z 60,A 168.9214,B 24.8201,C -3.093,E1 24.8401,E2 -806.2537} C_DIS
LIN {X -25.4303,Y 0.3624,Z 60,A 172.6307,B 24.8217,C -3.0796,E1 24.8398,E2 -809.9532} C_DIS
LIN {X -25.4197,Y -0.8106,Z 60,A 175.9195,B 24.8223,C -3.0749,E1 24.84,E2 -813.2504} C_DIS
LIN {X -25.1904,Y -3.5025,Z 60,A -178.4835,B 24.8247,C -3.0535,E1 24.8417,E2 -818.8297} C_DIS
LIN {X -24.8644,Y -5.3449,Z 60,A -173.8983,B 24.826,C -3.0428,E1 24.8441,E2 -823.4165} C_DIS
LIN {X -24.4853,Y -6.8752,Z 60,A -170.9034,B 24.8275,C -3.0292,E1 24.8462,E2 -826.3963} C_DIS
LIN {X -24.0787,Y -8.1876,Z 60,A -167.0599,B 24.8281,C -3.0245,E1 24.8496,E2 -830.2504} C_DIS
LIN {X -23.2645,Y -10.2749,Z 60,A -162.5228,B 24.83,C -3.0074,E1 24.8544,E2 -834.7719} C_DIS
LIN {X -22.6465,Y -11.574,Z 60,A -159.2581,B 24.831,C -2.9988,E1 24.8584,E2 -838.0335} C_DIS
LIN {X -21.7815,Y -13.1299,Z 60,A -154.7797,B 24.8318,C -2.9912,E1 24.8647,E2 -842.5171} C_DIS
LIN {X -20.8485,Y -14.5659,Z 60,A -151.3574,B 24.8332,C -2.9791,E1 24.87,E2 -845.9273} C_DIS
LIN {X -20.0047,Y -15.7042,Z 60,A -148.0683,B 24.834,C -2.9722,E1 24.8756,E2 -849.2156} C_DIS
LIN {X -19.0672,Y -16.8306,Z 60,A -144.8459,B 24.8349,C -2.9643,E1 24.8815,E2 -852.434} C_DIS
LIN {X -18.1283,Y -17.8377,Z 60,A -141.4097,B 24.8353,C -2.96,E1 24.8881,E2 -855.8746} C_DIS
LIN {X -16.9961,Y -18.9197,Z 60,A -138.3294,B 24.8364,C -2.9501,E1 24.8944,E2 -858.9439} C_DIS
LIN {X -15.4509,Y -20.2013,Z 60,A -132.6038,B 24.8364,C -2.9503,E1 24.907,E2 -864.6913} C_DIS
LIN {X -13.4851,Y -21.5632,Z 60,A -127.5948,B 24.8376,C -2.9395,E1 24.9187,E2 -869.6906} C_DIS
LIN {X -11.4144,Y -22.7277,Z 60,A -122.5429,B 24.8386,C -2.9305,E1 24.9311,E2 -874.7351} C_DIS
LIN {X -9.6542,Y -23.5289,Z 60,A -118.1868,B 24.8391,C -2.926,E1 24.9423,E2 -879.0907} C_DIS
LIN {X -7.9105,Y -24.1709,Z 60,A -113.9471,B 24.8394,C -2.923,E1 24.9534,E2 -883.3316} C_DIS
LIN {X -6.2662,Y -24.6482,Z 60,A -110.3455,B 24.8399,C -2.9187,E1 24.9631,E2 -886.9283} C_DIS
LIN {X -4.7195,Y -24.9908,Z 60,A -106.5999,B 24.8399,C -2.9187,E1 24.9734,E2 -890.6783} C_DIS
LIN {X -3.1936,Y -25.2314,Z 60,A -102.981,B 24.8399,C -2.9191,E1 24.9834,E2 -894.3011} C_DIS
LIN {X -1.2098,Y -25.4035,Z 60,A -98.6366,B 24.84,C -2.918,E1 24.9955,E2 -898.6443} C_DIS
LIN {X 0.0483,Y -25.4277,Z 60,A -96.2758,B 24.8404,C -2.9145,E1 25.0021,E2 -900.9968} C_DIS
Enddeposition()
LIN {X 0.0483,Y -25.4277,Z 60,A -96.2758,B 24.8404,C -2.9145,E1 25.0021,E2 -900.9968} C_DIS
Startdeposition()
$VEL.CP = VEL_PRINT
LIN {X -0.1194,Y -24.4743,Z 60,A -97.9411,B 24.8398,C -2.9201,E1 24.9975,E2 -899.3449} C_DIS
LIN {X -1.3912,Y -24.4345,Z 60,A -101.1551,B 24.84,C -2.9179,E1 24.9885,E2 -896.1251} C_DIS
LIN {X -3.0318,Y -24.2861,Z 60,A -105.2121,B 24.8401,C -2.9168,E1 24.9772,E2 -892.0628} C_DIS
LIN {X -5.1261,Y -23.9314,Z 60,A -109.3027,B 24.8392,C -2.9253,E1 24.966,E2 -887.9882} C_DIS
LIN {X -6.2048,Y -23.6747,Z 60,A -113.1473,B 24.8401,C -2.9174,E1 24.9556,E2 -884.1193} C_DIS
LIN {X -8.5961,Y -22.9147,Z 60,A -118.265,B 24.839,C -2.9275,E1 24.9421,E2 -879.0159} C_DIS
LIN {X -9.8621,Y -22.3995,Z 60,A -121.5676,B 24.8387,C -2.93,E1 24.9336,E2 -875.7117} C_DIS
LIN {X -11.22,Y -21.7514,Z 60,A -125.2921,B 24.8384,C -2.9328,E1 24.9242,E2 -871.984} C_DIS
LIN {X -13.0488,Y -20.7059,Z 60,A -130.3145,B 24.8377,C -2.9391,E1 24.9122,E2 -866.9614} C_DIS
LIN {X -14.4195,Y -19.7754,Z 60,A -134.1248,B 24.8369,C -2.9458,E1 24.9035,E2 -863.154} C_DIS
LIN {X -15.9092,Y -18.5985,Z 60,A -138.3748,B 24.8359,C -2.955,E1 24.8943,E2 -858.9099} C_DIS
LIN {X -17.0618,Y -17.5473,Z 60,A -142.1876,B 24.8352,C -2.9612,E1 24.8866,E2 -855.0964} C_DIS
LIN {X -18.0158,Y -16.5661,Z 60,A -145.0807,B 24.8342,C -2.9698,E1 24.8811,E2 -852.2113} C_DIS
LIN {X -18.8956,Y -15.5549,Z 60,A -148.6815,B 24.8338,C -2.9742,E1 24.8746,E2 -848.6045} C_DIS
LIN {X -20.0551,Y -14.0282,Z 60,A -153.0183,B 24.8325,C -2.9858,E1 24.8674,E2 -844.2743} C_DIS
LIN {X -20.8051,Y -12.8903,Z 60,A -155.9809,B 24.8314,C -2.995,E1 24.863,E2 -841.3188} C_DIS
LIN {X -21.7036,Y -11.3115,Z 60,A -161.0461,B 24.8306,C -3.0019,E1 24.8562,E2 -836.2434} C_DIS
LIN {X -22.5301,Y -9.5596,Z 60,A -165.0501,B 24.8289,C -3.0171,E1 24.8516,E2 -832.2539} C_DIS
LIN {X -23.041,Y -8.2526,Z 60,A -168.2987,B 24.8278,C -3.0266,E1 24.8485,E2 -829.0097} C_DIS
LIN {X -23.4063,Y -7.1512,Z 60,A -171.3662,B 24.8271,C -3.0328,E1 24.8459,E2 -825.9394} C_DIS
LIN {X -23.8975,Y -5.2809,Z 60,A -175.8045,B 24.8255,C -3.0467,E1 24.843,E2 -821.5084} C_DIS
LIN {X -24.2247,Y -3.4877,Z 60,A -179.6518,B 24.8238,C -3.0617,E1 24.8412,E2 -817.6742} C_DIS
LIN {X -24.4232,Y -1.5817,Z 60,A 175.3399,B 24.8225,C -3.073,E1 24.8399,E2 -812.663} C_DIS
LIN {X -24.4729,Y 0.188,Z 60,A 171.1822,B 24.821,C -3.0859,E1 24.8399,E2 -808.511} C_DIS
LIN {X -24.3806,Y 2.1408,Z 60,A 166.1022,B 24.8196,C -3.0978,E1 24.8408,E2 -803.4289} C_DIS
LIN {X -24.1062,Y 4.2316,Z 60,A 160.7606,B 24.818,C -3.1112,E1 24.8432,E2 -798.0878} C_DIS
LIN {X -23.2809,Y 7.5494,Z 60,A 154.1181,B 24.8143,C -3.1422,E1 24.848,E2 -791.481} C_DIS
LIN {X -22.8687,Y 8.7191,Z 60,A 150.5192,B 24.8137,C -3.1475,E1 24.8515,E2 -787.8745} C_DIS
LIN {X -22.1335,Y 10.4464,Z 60,A 146.5775,B 24.8119,C -3.1626,E1 24.8559,E2 -783.9472} C_DIS
LIN {X -21.6726,Y 11.3705,Z 60,A 143.8851,B 24.8113,C -3.1681,E1 24.8594,E2 -781.2537} C_DIS
LIN {X -20.9138,Y 12.7129,Z 60,A 139.94,B 24.8103,C -3.1765,E1 24.865,E2 -777.3082} C_DIS
LIN {X -19.6561,Y 14.5828,Z 60,A 134.6245,B 24.8086,C -3.1903,E1 24.8735,E2 -771.9997} C_DIS
LIN {X -18.5767,Y 15.9346,Z 60,A 131.1707,B 24.807,C -3.2037,E1 24.8796,E2 -768.562} C_DIS
LIN {X -17.9058,Y 16.6849,Z 60,A 128.1439,B 24.8067,C -3.2058,E1 24.8854,E2 -765.5268} C_DIS
LIN {X -16.2596,Y 18.2929,Z 60,A 123.0909,B 24.805,C -3.2199,E1 24.8956,E2 -760.4869} C_DIS
LIN {X -14.8657,Y 19.4422,Z 60,A 118.7188,B 24.804,C -3.2279,E1 24.9052,E2 -756.1177} C_DIS
LIN {X -13.3414,Y 20.5183,Z 60,A 114.034,B 24.8032,C -3.2344,E1 24.916,E2 -751.4327} C_DIS
LIN {X -11.5533,Y 21.5761,Z 60,A 109.8812,B 24.8017,C -3.247,E1 24.926,E2 -747.298} C_DIS
LIN {X -10.6178,Y 22.0512,Z 60,A 107.193,B 24.8014,C -3.2494,E1 24.9328,E2 -744.6083} C_DIS
LIN {X -9.4776,Y 22.5647,Z 60,A 103.7313,B 24.8014,C -3.25,E1 24.9417,E2 -741.1401} C_DIS
LIN {X -7.7429,Y 23.2169,Z 60,A 99.9799,B 24.8002,C -3.2593,E1 24.9515,E2 -737.4033} C_DIS
LIN {X -6.3092,Y 23.6469,Z 60,A 96.2215,B 24.8,C -3.2611,E1 24.9616,E2 -733.6435} C_DIS
LIN {X -4.8816,Y 23.9825,Z 60,A 93.0317,B 24.7994,C -3.2658,E1 24.9703,E2 -730.4607} C_DIS
LIN {X -3.6584,Y 24.1997,Z 60,A 90.1487,B 24.7991,C -3.268,E1 24.9782,E2 -727.5803} C_DIS
LIN {X -2.2491,Y 24.3708,Z 60,A 86.54,B 24.7991,C -3.2676,E1 24.9882,E2 -723.9685} C_DIS
LIN {X -0.7424,Y 24.4631,Z 60,A 83.2524,B 24.7988,C -3.2707,E1 24.9974,E2 -720.6874} C_DIS
LIN {X 1.2545,Y 24.442,Z 60,A 77.5299,B 24.7997,C -3.263,E1 25.0134,E2 -714.948} C_DIS
LIN {X 4.3435,Y 24.0857,Z 60,A 70.5758,B 24.7997,C -3.2638,E1 25.0326,E2 -708.002} C_DIS
LIN {X 6.2321,Y 23.6673,Z 60,A 66.6562,B 24.7993,C -3.2665,E1 25.0432,E2 -704.0943} C_DIS
LIN {X 7.6143,Y 23.2597,Z 60,A 63.3075,B 24.7996,C -3.2642,E1 25.0521,E2 -700.7463} C_DIS
LIN {X 8.9914,Y 22.7628,Z 60,A 59.7338,B 24.8001,C -3.2597,E1 25.0614,E2 -697.1697} C_DIS
LIN {X 10.4797,Y 22.1175,Z 60,A 55.9175,B 24.8007,C -3.2554,E1 25.0712,E2 -693.3525} C_DIS
LIN {X 12.4856,Y 21.0503,Z 60,A 50.0364,B 24.8022,C -3.243,E1 25.0855,E2 -687.4594} C_DIS
LIN {X 14.1227,Y 19.9887,Z 60,A 46.2635,B 24.8022,C -3.2433,E1 25.0942,E2 -683.6998} C_DIS
LIN {X 15.2853,Y 19.1146,Z 60,A 42.7805,B 24.803,C -3.2365,E1 25.1019,E2 -680.2137} C_DIS
LIN {X 16.4044,Y 18.1633,Z 60,A 39.5223,B 24.8036,C -3.2318,E1 25.1087,E2 -676.957} C_DIS
LIN {X 17.334,Y 17.2783,Z 60,A 36.5747,B 24.8042,C -3.2262,E1 25.1146,E2 -674.0087} C_DIS
LIN {X 18.1703,Y 16.3964,Z 60,A 33.2922,B 24.8055,C -3.2157,E1 25.1208,E2 -670.7155} C_DIS
LIN {X 19.7915,Y 14.3976,Z 60,A 26.2858,B 24.8084,C -3.1915,E1 25.1328,E2 -663.6851} C_DIS
LIN {X 21.6246,Y 11.4619,Z 60,A 18.8685,B 24.8101,C -3.1777,E1 25.1432,E2 -656.2732} C_DIS
LIN {X 22.5311,Y 9.5574,Z 60,A 14.2399,B 24.8113,C -3.1674,E1 25.1484,E2 -651.6453} C_DIS
LIN {X 23.2332,Y 7.6941,Z 60,A 9.782,B 24.8127,C -3.1562,E1 25.1526,E2 -647.1859} C_DIS
LIN {X 23.7565,Y 5.883,Z 60,A 5.6361,B 24.8139,C -3.1461,E1 25.1556,E2 -643.0399} C_DIS
LIN {X 24.0582,Y 4.4944,Z 60,A 2.3026,B 24.8151,C -3.136,E1 25.1575,E2 -639.7019} C_DIS
LIN {X 24.2893,Y 3.0049,Z 60,A -1.3745,B 24.8166,C -3.1235,E1 25.1589,E2 -636.017} C_DIS
LIN {X 24.4449,Y 1.1962,Z 60,A -5.6679,B 24.8182,C -3.1099,E1 25.1597,E2 -631.7167} C_DIS
LIN {X 24.4729,Y -0.2554,Z 60,A -8.5257,B 24.8187,C -3.1053,E1 25.1597,E2 -628.8651} C_DIS
LIN {X 24.3904,Y -2.0236,Z 60,A -13.6723,B 24.8215,C -3.0812,E1 25.1588,E2 -623.6921} C_DIS
LIN {X 24.1497,Y -3.9746,Z 60,A -17.7505,B 24.8225,C -3.0727,E1 25.1571,E2 -619.6176} C_DIS
LIN {X 23.7949,Y -5.7258,Z 60,A -21.8941,B 24.824,C -3.0602,E1 25.1546,E2 -615.4685} C_DIS
LIN {X 23.3307,Y -7.3933,Z 60,A -25.6849,B 24.8251,C -3.0507,E1 25.1516,E2 -611.6768} C_DIS
LIN {X 22.8681,Y -8.7211,Z 60,A -28.9058,B 24.8261,C -3.0416,E1 25.1485,E2 -608.4523} C_DIS
LIN {X 22.3045,Y -10.075,Z 60,A -32.4969,B 24.8275,C -3.0297,E1 25.1445,E2 -604.8528} C_DIS
LIN {X 21.4953,Y -11.7028,Z 60,A -36.4924,B 24.8285,C -3.0203,E1 25.1394,E2 -600.8562} C_DIS
LIN {X 20.8343,Y -12.8429,Z 60,A -39.5289,B 24.8295,C -3.0122,E1 25.1351,E2 -597.8161} C_DIS
LIN {X 20.1539,Y -13.8862,Z 60,A -42.8355,B 24.8308,C -3.0001,E1 25.1299,E2 -594.4972} C_DIS
LIN {X 18.918,Y -15.5278,Z 60,A -47.0176,B 24.8315,C -2.9943,E1 25.1227,E2 -590.321} C_DIS
LIN {X 17.7066,Y -16.8961,Z 60,A -52.0039,B 24.8335,C -2.9764,E1 25.1133,E2 -585.3143} C_DIS
LIN {X 16.2302,Y -18.3187,Z 60,A -56.3917,B 24.8343,C -2.9697,E1 25.1043,E2 -580.9283} C_DIS
LIN {X 15.0197,Y -19.3241,Z 60,A -59.9692,B 24.835,C -2.9629,E1 25.0965,E2 -577.3482} C_DIS
LIN {X 13.7016,Y -20.2798,Z 60,A -64.0392,B 24.8362,C -2.9528,E1 25.0872,E2 -573.2683} C_DIS
LIN {X 12.4849,Y -21.0507,Z 60,A -66.9201,B 24.8362,C -2.9514,E1 25.0804,E2 -570.3934} C_DIS
LIN {X 11.3572,Y -21.6796,Z 60,A -70.22,B 24.8372,C -2.9437,E1 25.0722,E2 -567.0844} C_DIS
LIN {X 9.8422,Y -22.4081,Z 60,A -74.3194,B 24.838,C -2.9361,E1 25.0618,E2 -562.9776} C_DIS
LIN {X 8.2161,Y -23.054,Z 60,A -78.0869,B 24.8383,C -2.9338,E1 25.052,E2 -559.2126} C_DIS
LIN {X 7.1091,Y -23.4191,Z 60,A -80.8396,B 24.8386,C -2.9304,E1 25.0447,E2 -556.457} C_DIS
LIN {X 5.8215,Y -23.7714,Z 60,A -83.7867,B 24.8388,C -2.9289,E1 25.0367,E2 -553.5108} C_DIS
LIN {X 4.7418,Y -24.0109,Z 60,A -86.6811,B 24.8393,C -2.924,E1 25.0288,E2 -550.6083} C_DIS
LIN {X 3.0824,Y -24.2793,Z 60,A -90.16,B 24.8393,C -2.9252,E1 25.0192,E2 -547.1356} C_DIS
LIN {X 1.1313,Y -24.4478,Z 60,A -95.6966,B 24.8403,C -2.9152,E1 25.0037,E2 -541.5776} C_DIS
LIN {X 1.1313,Y -24.4478,Z 60,A -95.6966,B 24.8403,C -2.9152,E1 25.0037,E2 -541.5776} C_DIS
Enddeposition()
LIN {X 0.042,Y -23.5166,Z 60,A -95.9371,B 24.8365,C -2.9501,E1 25.0033,E2 -541.4202} C_DIS
Startdeposition()
$VEL.CP = VEL_PRINT
LIN {X 1.6328,Y -23.4591,Z 60,A -91.9005,B 24.8361,C -2.9529,E1 25.0145,E2 -545.4621} C_DIS
LIN {X 3.3721,Y -23.2734,Z 60,A -87.4627,B 24.8357,C -2.9571,E1 25.0268,E2 -549.9063} C_DIS
LIN {X 5.3316,Y -22.904,Z 60,A -83.0234,B 24.8357,C -2.9576,E1 25.039,E2 -554.3411} C_DIS
LIN {X 6.8001,Y -22.5118,Z 60,A -79.0203,B 24.8349,C -2.9643,E1 25.0497,E2 -558.3534} C_DIS
LIN {X 8.5261,Y -21.916,Z 60,A -74.8482,B 24.8345,C -2.9674,E1 25.0607,E2 -562.5243} C_DIS
LIN {X 9.9592,Y -21.3032,Z 60,A -70.672,B 24.8335,C -2.9767,E1 25.0713,E2 -566.712} C_DIS
LIN {X 11.904,Y -20.2811,Z 60,A -66.1282,B 24.8333,C -2.9779,E1 25.0824,E2 -571.2457} C_DIS
LIN {X 13.3897,Y -19.3321,Z 60,A -60.9749,B 24.8315,C -2.9946,E1 25.0945,E2 -576.4215} C_DIS
LIN {X 14.7464,Y -18.3185,Z 60,A -57.5404,B 24.8313,C -2.9963,E1 25.102,E2 -579.8473} C_DIS
LIN {X 15.7406,Y -17.4716,Z 60,A -54.2831,B 24.8304,C -3.0041,E1 25.1089,E2 -583.1103} C_DIS
LIN {X 16.8849,Y -16.3682,Z 60,A -50.0494,B 24.8289,C -3.017,E1 25.1172,E2 -587.3567} C_DIS
LIN {X 17.9383,Y -15.2067,Z 60,A -46.1508,B 24.8277,C -3.0274,E1 25.1244,E2 -591.2623} C_DIS
LIN {X 19.2822,Y -13.4616,Z 60,A -41.5745,B 24.8271,C -3.0332,E1 25.132,E2 -595.8303} C_DIS
LIN {X 20.1997,Y -12.0417,Z 60,A -36.6076,B 24.8247,C -3.0536,E1 25.1394,E2 -600.8205} C_DIS
LIN {X 21.0213,Y -10.5422,Z 60,A -32.5736,B 24.8235,C -3.0642,E1 25.1445,E2 -604.8581} C_DIS
LIN {X 21.8799,Y -8.6186,Z 60,A -27.743,B 24.8221,C -3.0761,E1 25.1498,E2 -609.6904} C_DIS
LIN {X 22.3514,Y -7.3094,Z 60,A -24.757,B 24.8214,C -3.0819,E1 25.1525,E2 -612.6734} C_DIS
LIN {X 22.6826,Y -6.2062,Z 60,A -21.8331,B 24.8203,C -3.0918,E1 25.1547,E2 -615.6039} C_DIS
LIN {X 22.9602,Y -5.0841,Z 60,A -18.6424,B 24.8188,C -3.1046,E1 25.1567,E2 -618.8064} C_DIS
LIN {X 23.3072,Y -3.128,Z 60,A -13.6211,B 24.8168,C -3.1217,E1 25.1588,E2 -623.8386} C_DIS
LIN {X 23.4984,Y -0.914,Z 60,A -8.8391,B 24.8156,C -3.1316,E1 25.1597,E2 -628.6158} C_DIS
LIN {X 23.5123,Y 0.4405,Z 60,A -5.389,B 24.8142,C -3.1435,E1 25.1597,E2 -632.0736} C_DIS
LIN {X 23.4327,Y 1.9793,Z 60,A -1.3717,B 24.8125,C -3.158,E1 25.1589,E2 -636.1015} C_DIS
LIN {X 23.1361,Y 4.2121,Z 60,A 3.8872,B 24.8108,C -3.1722,E1 25.1566,E2 -641.3631} C_DIS
LIN {X 22.6361,Y 6.3724,Z 60,A 9.5965,B 24.8084,C -3.1916,E1 25.1527,E2 -647.0854} C_DIS
LIN {X 22.0583,Y 8.1507,Z 60,A 13.5865,B 24.8076,C -3.1986,E1 25.149,E2 -651.0696} C_DIS
LIN {X 21.523,Y 9.4755,Z 60,A 17.0295,B 24.8065,C -3.2079,E1 25.1453,E2 -654.5157} C_DIS
LIN {X 20.9662,Y 10.651,Z 60,A 20.0652,B 24.8056,C -3.2151,E1 25.1415,E2 -657.5521} C_DIS
LIN {X 20.4472,Y 11.6161,Z 60,A 23.1038,B 24.8043,C -3.2259,E1 25.1374,E2 -660.6007} C_DIS
LIN {X 19.4864,Y 13.1637,Z 60,A 27.7734,B 24.8026,C -3.2395,E1 25.1302,E2 -665.279} C_DIS
LIN {X 18.1279,Y 14.9802,Z 60,A 32.685,B 24.8018,C -3.246,E1 25.1218,E2 -670.1831} C_DIS
LIN {X 17.0131,Y 16.2353,Z 60,A 37.2269,B 24.8002,C -3.2594,E1 25.1132,E2 -674.7367} C_DIS
LIN {X 15.7211,Y 17.4892,Z 60,A 41.0437,B 24.7998,C -3.2625,E1 25.1054,E2 -678.5452} C_DIS
LIN {X 14.8065,Y 18.2699,Z 60,A 44.1078,B 24.799,C -3.2692,E1 25.0988,E2 -681.6135} C_DIS
LIN {X 13.5922,Y 19.1902,Z 60,A 47.862,B 24.7981,C -3.2758,E1 25.0904,E2 -685.3701} C_DIS
LIN {X 12.1761,Y 20.1187,Z 60,A 52.0486,B 24.7973,C -3.2825,E1 25.0805,E2 -689.5593} C_DIS
LIN {X 10.7531,Y 20.9133,Z 60,A 56.3483,B 24.7963,C -3.2907,E1 25.0699,E2 -693.8661} C_DIS
LIN {X 8.8963,Y 21.7685,Z 60,A 61.2682,B 24.7957,C -3.2954,E1 25.0573,E2 -698.7854} C_DIS
LIN {X 6.9814,Y 22.4559,Z 60,A 65.9674,B 24.7955,C -3.2971,E1 25.0448,E2 -703.4797} C_DIS
LIN {X 5.392,Y 22.8898,Z 60,A 69.9245,B 24.7953,C -3.299,E1 25.0341,E2 -707.4352} C_DIS
LIN {X 3.8029,Y 23.207,Z 60,A 73.5652,B 24.7953,C -3.2979,E1 25.0241,E2 -711.0693} C_DIS
LIN {X 2.28,Y 23.4055,Z 60,A 77.1154,B 24.7955,C -3.2971,E1 25.0143,E2 -714.6149} C_DIS
LIN {X 0.8118,Y 23.5024,Z 60,A 81.4968,B 24.7947,C -3.3031,E1 25.0021,E2 -719.0092} C_DIS
LIN {X -1.2435,Y 23.4831,Z 60,A 86.3449,B 24.7951,C -3.3005,E1 24.9885,E2 -723.8517} C_DIS
LIN {X -3.3756,Y 23.2729,Z 60,A 91.7191,B 24.7953,C -3.2986,E1 24.9737,E2 -729.2252} C_DIS
LIN {X -5.3029,Y 22.9106,Z 60,A 95.8938,B 24.7963,C -3.2905,E1 24.9623,E2 -733.3854} C_DIS
LIN {X -6.3149,Y 22.6522,Z 60,A 99.0759,B 24.7961,C -3.2923,E1 24.9537,E2 -736.5767} C_DIS
LIN {X -8.4272,Y 21.9543,Z 60,A 104.3596,B 24.797,C -3.2847,E1 24.9398,E2 -741.8528} C_DIS
LIN {X -10.2566,Y 21.1613,Z 60,A 108.7844,B 24.7983,C -3.2749,E1 24.9286,E2 -746.2649} C_DIS
LIN {X -11.3228,Y 20.6115,Z 60,A 111.9442,B 24.7987,C -3.2716,E1 24.9208,E2 -749.4255} C_DIS
LIN {X -12.6057,Y 19.8525,Z 60,A 115.3038,B 24.7997,C -3.2635,E1 24.9128,E2 -752.7762} C_DIS
LIN {X -13.4689,Y 19.2773,Z 60,A 118.1911,B 24.8,C -3.2607,E1 24.9062,E2 -755.6665} C_DIS
LIN {X -14.7642,Y 18.3037,Z 60,A 122.2027,B 24.801,C -3.2529,E1 24.8973,E2 -759.6743} C_DIS
LIN {X -15.9588,Y 17.2726,Z 60,A 126.109,B 24.802,C -3.2447,E1 24.8892,E2 -763.5765} C_DIS
LIN {X -17.2235,Y 16.0118,Z 60,A 130.1211,B 24.8035,C -3.2326,E1 24.8814,E2 -767.5768} C_DIS
LIN {X -17.9442,Y 15.1997,Z 60,A 133.2218,B 24.804,C -3.2284,E1 24.8758,E2 -770.6816} C_DIS
LIN {X -18.8129,Y 14.11,Z 60,A 136.3744,B 24.8052,C -3.2184,E1 24.8705,E2 -773.8252} C_DIS
LIN {X -19.6483,Y 12.9213,Z 60,A 139.6636,B 24.8065,C -3.2076,E1 24.8653,E2 -777.105} C_DIS
LIN {X -20.3432,Y 11.7976,Z 60,A 143.3367,B 24.8073,C -3.2009,E1 24.86,E2 -780.781} C_DIS
LIN {X -21.2028,Y 10.1713,Z 60,A 147.3266,B 24.8091,C -3.1857,E1 24.855,E2 -784.7558} C_DIS
LIN {X -21.7314,Y 8.9863,Z 60,A 151.4161,B 24.8097,C -3.1809,E1 24.8505,E2 -788.8564} C_DIS
LIN {X -22.4212,Y 7.0911,Z 60,A 156.1467,B 24.8116,C -3.1652,E1 24.8463,E2 -793.5764} C_DIS
LIN {X -22.922,Y 5.2534,Z 60,A 160.3295,B 24.8136,C -3.1488,E1 24.8434,E2 -797.7443} C_DIS
LIN {X -23.2167,Y 3.7444,Z 60,A 163.7748,B 24.8151,C -3.1358,E1 24.8417,E2 -801.1788} C_DIS
LIN {X -23.4039,Y 2.2968,Z 60,A 168.3087,B 24.8159,C -3.1293,E1 24.8402,E2 -805.7243} C_DIS
LIN {X -23.506,Y 0.6899,Z 60,A 172.073,B 24.8174,C -3.1163,E1 24.8398,E2 -809.4801} C_DIS
LIN {X -23.4908,Y -1.0913,Z 60,A 175.9821,B 24.8192,C -3.1008,E1 24.8401,E2 -813.3757} C_DIS
LIN {X -23.3826,Y -2.5035,Z 60,A 179.761,B 24.8203,C -3.0917,E1 24.841,E2 -817.1554} C_DIS
LIN {X -23.1251,Y -4.2707,Z 60,A -175.2191,B 24.8215,C -3.0817,E1 24.8434,E2 -822.1813} C_DIS
LIN {X -22.6197,Y -6.4293,Z 60,A -169.9323,B 24.8234,C -3.0652,E1 24.8471,E2 -827.4592} C_DIS
LIN {X -21.8537,Y -8.6848,Z 60,A -164.5166,B 24.8255,C -3.0467,E1 24.8523,E2 -832.8612} C_DIS
LIN {X -20.7642,Y -11.0391,Z 60,A -156.9116,B 24.8267,C -3.0364,E1 24.8618,E2 -840.4825} C_DIS
LIN {X -19.1271,Y -13.6808,Z 60,A -150.382,B 24.8295,C -3.0119,E1 24.8718,E2 -846.9862} C_DIS
LIN {X -18.1505,Y -14.9527,Z 60,A -146.7904,B 24.8307,C -3.0012,E1 24.878,E2 -850.5689} C_DIS
LIN {X -17.1425,Y -16.0983,Z 60,A -142.5019,B 24.8312,C -2.9965,E1 24.8861,E2 -854.8651} C_DIS
LIN {X -15.3247,Y -17.8376,Z 60,A -136.7446,B 24.8328,C -2.9823,E1 24.898,E2 -860.6119} C_DIS
LIN {X -13.6397,Y -19.1566,Z 60,A -130.606,B 24.8332,C -2.9794,E1 24.9117,E2 -866.7652} C_DIS
LIN {X -11.6198,Y -20.445,Z 60,A -125.424,B 24.8346,C -2.9668,E1 24.9241,E2 -871.9331} C_DIS
LIN {X -9.7753,Y -21.3882,Z 60,A -120.7132,B 24.8355,C -2.9587,E1 24.9359,E2 -876.6366} C_DIS
LIN {X -8.4065,Y -21.9627,Z 60,A -116.6629,B 24.8355,C -2.9583,E1 24.9465,E2 -880.6949} C_DIS
LIN {X -6.4258,Y -22.6208,Z 60,A -111.7838,B 24.8361,C -2.9532,E1 24.9595,E2 -885.5704} C_DIS
LIN {X -4.0716,Y -23.1611,Z 60,A -105.4933,B 24.8361,C -2.9539,E1 24.9767,E2 -891.8698} C_DIS
LIN {X -2.242,Y -23.4091,Z 60,A -101.6103,B 24.8366,C -2.9485,E1 24.9874,E2 -895.7424} C_DIS
LIN {X -0.7526,Y -23.5043,Z 60,A -97.881,B 24.8366,C -2.9495,E1 24.9978,E2 -899.475} C_DIS
LIN {X -0.7526,Y -23.5043,Z 60,A -97.881,B 24.8366,C -2.9495,E1 24.9978,E2 -899.475} C_DIS
Enddeposition()
LIN {X 0.0549,Y -22.5554,Z 60,A -97.7707,B 24.8362,C -2.9519,E1 24.9982,E2 -899.5912} C_DIS
Startdeposition()
$VEL.CP = VEL_PRINT
LIN {X -1.7553,Y -22.4894,Z 60,A -102.013,B 24.836,C -2.9543,E1 24.9863,E2 -895.3532} C_DIS
LIN {X -2.7082,Y -22.3949,Z 60,A -105.0789,B 24.8365,C -2.95,E1 24.9778,E2 -892.2752} C_DIS
LIN {X -4.5934,Y -22.085,Z 60,A -109.3144,B 24.8358,C -2.9559,E1 24.9662,E2 -888.0496} C_DIS
LIN {X -5.5323,Y -21.869,Z 60,A -112.6033,B 24.8363,C -2.9515,E1 24.9572,E2 -884.7455} C_DIS
LIN {X -7.727,Y -21.193,Z 60,A -118.1808,B 24.8356,C -2.9576,E1 24.9425,E2 -879.1723} C_DIS
LIN {X -9.8368,Y -20.3004,Z 60,A -124.3169,B 24.8351,C -2.9619,E1 24.9268,E2 -873.0315} C_DIS
LIN {X -11.6032,Y -19.3458,Z 60,A -129.9763,B 24.8347,C -2.9656,E1 24.9131,E2 -867.364} C_DIS
LIN {X -13.9464,Y -17.7298,Z 60,A -136.1813,B 24.8327,C -2.9833,E1 24.8992,E2 -861.1796} C_DIS
LIN {X -14.983,Y -16.8631,Z 60,A -140.1686,B 24.8323,C -2.9868,E1 24.8908,E2 -857.1849} C_DIS
LIN {X -16.6468,Y -15.2237,Z 60,A -145.3832,B 24.8305,C -3.0028,E1 24.8806,E2 -851.9863} C_DIS
LIN {X -17.5814,Y -14.1342,Z 60,A -149.3312,B 24.8298,C -3.0095,E1 24.8736,E2 -848.0361} C_DIS
LIN {X -18.4949,Y -12.9153,Z 60,A -152.9311,B 24.8286,C -3.0201,E1 24.8677,E2 -844.444} C_DIS
LIN {X -19.109,Y -11.9885,Z 60,A -156.5186,B 24.8282,C -3.0235,E1 24.8623,E2 -840.8467} C_DIS
LIN {X -20.209,Y -10.0222,Z 60,A -161.6073,B 24.8261,C -3.0416,E1 24.8556,E2 -835.7742} C_DIS
LIN {X -20.8905,Y -8.5114,Z 60,A -166.1031,B 24.8249,C -3.052,E1 24.8506,E2 -831.2785} C_DIS
LIN {X -21.505,Y -6.8109,Z 60,A -170.9622,B 24.8235,C -3.064,E1 24.8463,E2 -826.4205} C_DIS
LIN {X -21.9837,Y -5.0579,Z 60,A -175.5546,B 24.8219,C -3.0778,E1 24.8432,E2 -821.8343} C_DIS
LIN {X -22.3407,Y -3.1252,Z 60,A 179.7434,B 24.82,C -3.0942,E1 24.841,E2 -817.1437} C_DIS
LIN {X -22.4998,Y -1.6175,Z 60,A 175.6441,B 24.8187,C -3.105,E1 24.84,E2 -813.0457} C_DIS
LIN {X -22.556,Y -0.3336,Z 60,A 172.6571,B 24.8174,C -3.1163,E1 24.8398,E2 -810.0678} C_DIS
LIN {X -22.5203,Y 1.3017,Z 60,A 168.092,B 24.8161,C -3.1276,E1 24.8403,E2 -805.5022} C_DIS
LIN {X -22.3586,Y 2.9943,Z 60,A 163.8563,B 24.8144,C -3.1414,E1 24.8416,E2 -801.2741} C_DIS
LIN {X -22.0806,Y 4.6182,Z 60,A 159.6314,B 24.8129,C -3.1542,E1 24.8438,E2 -797.0549} C_DIS
LIN {X -21.6804,Y 6.23,Z 60,A 155.3891,B 24.8114,C -3.167,E1 24.8469,E2 -792.8186} C_DIS
LIN {X -21.2277,Y 7.632,Z 60,A 151.137,B 24.8103,C -3.1761,E1 24.8508,E2 -788.5642} C_DIS
LIN {X -20.5034,Y 9.406,Z 60,A 146.5389,B 24.8084,C -3.1915,E1 24.8559,E2 -783.9776} C_DIS
LIN {X -19.4334,Y 11.4552,Z 60,A 140.3971,B 24.8066,C -3.2069,E1 24.8642,E2 -777.8403} C_DIS
LIN {X -18.2083,Y 13.3167,Z 60,A 134.6564,B 24.8048,C -3.2216,E1 24.8733,E2 -772.1067} C_DIS
LIN {X -16.7805,Y 15.0761,Z 60,A 129.4064,B 24.8028,C -3.2384,E1 24.8828,E2 -766.8728} C_DIS
LIN {X -15.4601,Y 16.4273,Z 60,A 124.3764,B 24.8015,C -3.2484,E1 24.8928,E2 -761.8456} C_DIS
LIN {X -14.009,Y 17.6807,Z 60,A 119.1858,B 24.8004,C -3.2571,E1 24.9039,E2 -756.6563} C_DIS
LIN {X -12.8323,Y 18.553,Z 60,A 115.1071,B 24.7998,C -3.2625,E1 24.9133,E2 -752.5765} C_DIS
LIN {X -10.6905,Y 19.8644,Z 60,A 109.5825,B 24.7978,C -3.2782,E1 24.9266,E2 -747.0728} C_DIS
LIN {X -9.3012,Y 20.5514,Z 60,A 105.6468,B 24.7971,C -3.2841,E1 24.9365,E2 -743.1414} C_DIS
LIN {X -8.1191,Y 21.0464,Z 60,A 102.0916,B 24.7968,C -3.2867,E1 24.9457,E2 -739.5845} C_DIS
LIN {X -6.3661,Y 21.6407,Z 60,A 98.1028,B 24.7956,C -3.2964,E1 24.9563,E2 -735.6117} C_DIS
LIN {X -5.1265,Y 21.968,Z 60,A 94.2601,B 24.7956,C -3.2957,E1 24.9667,E2 -731.7621} C_DIS
LIN {X -3.723,Y 22.249,Z 60,A 90.8899,B 24.7951,C -3.3002,E1 24.9759,E2 -728.3989} C_DIS
LIN {X -2.4741,Y 22.4223,Z 60,A 87.5541,B 24.795,C -3.3011,E1 24.9852,E2 -725.0631} C_DIS
LIN {X -1.0657,Y 22.5327,Z 60,A 84.1061,B 24.7947,C -3.3035,E1 24.9948,E2 -721.6195} C_DIS
LIN {X 0.3327,Y 22.556,Z 60,A 80.3888,B 24.7947,C -3.303,E1 25.0052,E2 -717.9012} C_DIS
LIN {X 1.7629,Y 22.489,Z 60,A 76.8367,B 24.7947,C -3.3037,E1 25.015,E2 -714.352} C_DIS
LIN {X 3.5954,Y 22.2698,Z 60,A 71.3497,B 24.7956,C -3.2966,E1 25.0302,E2 -708.853} C_DIS
LIN {X 5.577,Y 21.8576,Z 60,A 66.1341,B 24.796,C -3.2932,E1 25.0444,E2 -703.6369} C_DIS
LIN {X 7.9186,Y 21.1222,Z 60,A 60.9889,B 24.7955,C -3.297,E1 25.058,E2 -698.5105} C_DIS
LIN {X 8.9586,Y 20.7026,Z 60,A 56.7392,B 24.7973,C -3.2824,E1 25.0689,E2 -694.2363} C_DIS
LIN {X 11.7085,Y 19.2815,Z 60,A 49.9702,B 24.7975,C -3.2813,E1 25.0854,E2 -687.4844} C_DIS
LIN {X 13.4667,Y 18.0978,Z 60,A 44.203,B 24.799,C -3.2691,E1 25.0986,E2 -681.7081} C_DIS
LIN {X 15.0377,Y 16.815,Z 60,A 39.4605,B 24.7997,C -3.2632,E1 25.1087,E2 -676.9701} C_DIS
LIN {X 16.3774,Y 15.5133,Z 60,A 34.4936,B 24.8012,C -3.2513,E1 25.1185,E2 -671.996} C_DIS
LIN {X 17.4432,Y 14.3047,Z 60,A 30.9372,B 24.8017,C -3.2472,E1 25.1249,E2 -668.4462} C_DIS
LIN {X 18.1331,Y 13.4186,Z 60,A 27.9858,B 24.8026,C -3.2395,E1 25.1299,E2 -665.4906} C_DIS
LIN {X 18.972,Y 12.2041,Z 60,A 24.2543,B 24.8037,C -3.2304,E1 25.1357,E2 -661.756} C_DIS
LIN {X 19.8682,Y 10.6834,Z 60,A 19.3522,B 24.8057,C -3.2146,E1 25.1424,E2 -656.8418} C_DIS
LIN {X 20.7597,Y 8.8262,Z 60,A 14.4393,B 24.807,C -3.2034,E1 25.1481,E2 -651.929} C_DIS
LIN {X 21.3353,Y 7.3263,Z 60,A 10.1054,B 24.8087,C -3.1892,E1 25.1523,E2 -647.5856} C_DIS
LIN {X 21.9049,Y 5.3874,Z 60,A 5.9054,B 24.8094,C -3.1836,E1 25.1554,E2 -643.3966} C_DIS
LIN {X 22.1457,Y 4.2939,Z 60,A 1.8124,B 24.812,C -3.1622,E1 25.1577,E2 -639.2766} C_DIS
LIN {X 22.4844,Y 1.8213,Z 60,A -3.5903,B 24.8131,C -3.1524,E1 25.1594,E2 -633.8827} C_DIS
LIN {X 22.5497,Y 0.6159,Z 60,A -6.9737,B 24.8147,C -3.1396,E1 25.1598,E2 -630.489} C_DIS
LIN {X 22.5324,Y -1.0724,Z 60,A -10.8846,B 24.8158,C -3.1301,E1 25.1595,E2 -626.5791} C_DIS
LIN {X 22.4468,Y -2.2405,Z 60,A -13.9078,B 24.8169,C -3.1203,E1 25.1588,E2 -623.5505} C_DIS
LIN {X 22.2933,Y -3.4479,Z 60,A -17.2908,B 24.8184,C -3.1076,E1 25.1574,E2 -620.1573} C_DIS
LIN {X 21.9356,Y -5.262,Z 60,A -21.2043,B 24.8192,C -3.1013,E1 25.1552,E2 -616.2517} C_DIS
LIN {X 21.626,Y -6.4174,Z 60,A -24.6753,B 24.8208,C -3.0875,E1 25.1526,E2 -612.7678} C_DIS
LIN {X 21.2731,Y -7.5051,Z 60,A -27.33,B 24.8215,C -3.0813,E1 25.1502,E2 -610.1134} C_DIS
LIN {X 20.6598,Y -9.0576,Z 60,A -32.5834,B 24.8242,C -3.0583,E1 25.1445,E2 -604.8345} C_DIS
LIN {X 19.7264,Y -10.942,Z 60,A -37.4318,B 24.8254,C -3.048,E1 25.1382,E2 -599.9873} C_DIS
LIN {X 18.752,Y -12.5397,Z 60,A -41.5906,B 24.8262,C -3.0409,E1 25.132,E2 -595.8327} C_DIS
LIN {X 17.739,Y -13.9358,Z 60,A -46.2977,B 24.8279,C -3.0261,E1 25.1241,E2 -591.113} C_DIS
LIN {X 16.9259,Y -14.9129,Z 60,A -49.2066,B 24.8284,C -3.0212,E1 25.1188,E2 -588.2056} C_DIS
LIN {X 16.061,Y -15.8403,Z 60,A -52.6049,B 24.8295,C -3.0117,E1 25.1123,E2 -584.7995} C_DIS
LIN {X 14.8948,Y -16.9416,Z 60,A -57.0969,B 24.831,C -2.9984,E1 25.103,E2 -580.2942} C_DIS
LIN {X 13.6428,Y -17.9657,Z 60,A -60.8251,B 24.8316,C -2.9934,E1 25.0948,E2 -576.5678} C_DIS
LIN {X 12.4966,Y -18.7804,Z 60,A -64.1712,B 24.8321,C -2.9885,E1 25.0871,E2 -573.2215} C_DIS
LIN {X 11.5392,Y -19.3837,Z 60,A -67.8154,B 24.8335,C -2.9763,E1 25.0783,E2 -569.5596} C_DIS
LIN {X 9.2918,Y -20.5556,Z 60,A -74.2896,B 24.8347,C -2.9659,E1 25.0621,E2 -563.0779} C_DIS
LIN {X 7.1405,Y -21.3978,Z 60,A -79.3946,B 24.8347,C -2.9649,E1 25.0487,E2 -557.9812} C_DIS
LIN {X 5.5234,Y -21.8712,Z 60,A -83.9302,B 24.8355,C -2.9582,E1 25.0365,E2 -553.4373} C_DIS
LIN {X 3.9128,Y -22.2163,Z 60,A -87.9906,B 24.8358,C -2.9558,E1 25.0254,E2 -549.3759} C_DIS
LIN {X 2.4002,Y -22.4301,Z 60,A -91.9415,B 24.8361,C -2.9529,E1 25.0144,E2 -545.4211} C_DIS
LIN {X 0.5143,Y -22.5513,Z 60,A -96.3338,B 24.836,C -2.9542,E1 25.0022,E2 -541.0334} C_DIS
LIN {X 0.5143,Y -22.5513,Z 60,A -96.3338,B 24.836,C -2.9542,E1 25.0022,E2 -541.0334} C_DIS
Enddeposition()
LIN {X 0.0454,Y -21.5985,Z 60,A -96.4918,B 24.8333,C -2.9783,E1 25.0019,E2 -540.9329} C_DIS
Startdeposition()
$VEL.CP = VEL_PRINT
LIN {X 1.5529,Y -21.5438,Z 60,A -92.0862,B 24.8328,C -2.9829,E1 25.0142,E2 -545.3478} C_DIS
LIN {X 3.0329,Y -21.3861,Z 60,A -87.506,B 24.8319,C -2.9903,E1 25.0269,E2 -549.9422} C_DIS
LIN {X 5.3094,Y -20.9364,Z 60,A -81.9713,B 24.8319,C -2.9907,E1 25.042,E2 -555.4705} C_DIS
LIN {X 6.5557,Y -20.5808,Z 60,A -78.8426,B 24.8317,C -2.992,E1 25.0504,E2 -558.5966} C_DIS
LIN {X 7.7985,Y -20.143,Z 60,A -74.8704,B 24.8308,C -3.0006,E1 25.0608,E2 -562.5809} C_DIS
LIN {X 9.0239,Y -19.6245,Z 60,A -71.7285,B 24.8306,C -3.0024,E1 25.0688,E2 -565.7194} C_DIS
LIN {X 10.2189,Y -19.0302,Z 60,A -67.9387,B 24.8297,C -3.0104,E1 25.0782,E2 -569.5176} C_DIS
LIN {X 11.7446,Y -18.1281,Z 60,A -62.6319,B 24.8281,C -3.0245,E1 25.0909,E2 -574.8413} C_DIS
LIN {X 13.0427,Y -17.2181,Z 60,A -58.3502,B 24.827,C -3.0339,E1 25.1005,E2 -579.1297} C_DIS
LIN {X 14.8792,Y -15.6586,Z 60,A -52.9888,B 24.8265,C -3.0383,E1 25.1116,E2 -584.4804} C_DIS
LIN {X 15.598,Y -14.942,Z 60,A -50.0859,B 24.8255,C -3.0468,E1 25.1173,E2 -587.3909} C_DIS
LIN {X 16.6968,Y -13.704,Z 60,A -44.8657,B 24.8233,C -3.066,E1 25.1268,E2 -592.6329} C_DIS
LIN {X 18.0569,Y -11.854,Z 60,A -39.4653,B 24.8222,C -3.0754,E1 25.1354,E2 -598.0292} C_DIS
LIN {X 18.9762,Y -10.3184,Z 60,A -34.8369,B 24.8208,C -3.0876,E1 25.1418,E2 -602.6624} C_DIS
LIN {X 19.8491,Y -8.5183,Z 60,A -28.6868,B 24.8179,C -3.1118,E1 25.1489,E2 -608.8364} C_DIS
LIN {X 20.8335,Y -5.7003,Z 60,A -21.0403,B 24.8154,C -3.133,E1 25.1553,E2 -616.4898} C_DIS
LIN {X 21.2505,Y -3.8711,Z 60,A -16.9672,B 24.8147,C -3.139,E1 25.1576,E2 -620.5534} C_DIS
LIN {X 21.467,Y -2.3908,Z 60,A -12.3118,B 24.8124,C -3.1585,E1 25.1592,E2 -625.2275} C_DIS
LIN {X 21.5985,Y -0.1629,Z 60,A -6.7484,B 24.8106,C -3.1733,E1 25.1598,E2 -630.7929} C_DIS
LIN {X 21.5357,Y 1.6633,Z 60,A -1.9246,B 24.8089,C -3.1881,E1 25.159,E2 -635.623} C_DIS
LIN {X 21.3181,Y 3.4775,Z 60,A 2.3349,B 24.8078,C -3.1968,E1 25.1574,E2 -639.8782} C_DIS
LIN {X 21.1325,Y 4.4698,Z 60,A 5.731,B 24.8059,C -3.2123,E1 25.1555,E2 -643.2911} C_DIS
LIN {X 20.5778,Y 6.5645,Z 60,A 11.1372,B 24.8043,C -3.2256,E1 25.1513,E2 -648.698} C_DIS
LIN {X 20.132,Y 7.826,Z 60,A 15.1626,B 24.8025,C -3.2405,E1 25.1473,E2 -652.7364} C_DIS
LIN {X 19.1406,Y 10.0097,Z 60,A 21.128,B 24.8009,C -3.2538,E1 25.14,E2 -658.7012} C_DIS
LIN {X 18.2056,Y 11.6244,Z 60,A 25.2484,B 24.8003,C -3.2584,E1 25.1341,E2 -662.8115} C_DIS
LIN {X 17.4374,Y 12.7478,Z 60,A 29.9582,B 24.7979,C -3.2778,E1 25.1265,E2 -667.5443} C_DIS
LIN {X 15.9281,Y 14.5898,Z 60,A 36.0843,B 24.7964,C -3.29,E1 25.1153,E2 -673.6716} C_DIS
LIN {X 14.8104,Y 15.7231,Z 60,A 39.7033,B 24.796,C -3.293,E1 25.1081,E2 -677.2826} C_DIS
LIN {X 13.8474,Y 16.5776,Z 60,A 43.8251,B 24.7944,C -3.3058,E1 25.0993,E2 -681.4188} C_DIS
LIN {X 11.959,Y 17.9869,Z 60,A 49.115,B 24.7942,C -3.3076,E1 25.0873,E2 -686.6945} C_DIS
LIN {X 11.039,Y 18.5664,Z 60,A 52.0777,B 24.7936,C -3.3125,E1 25.0802,E2 -689.6595} C_DIS
LIN {X 9.5773,Y 19.3605,Z 60,A 57.7943,B 24.7915,C -3.329,E1 25.066,E2 -695.3996} C_DIS
LIN {X 7.7483,Y 20.1626,Z 60,A 62.1649,B 24.7918,C -3.3266,E1 25.0547,E2 -699.7546} C_DIS
LIN {X 6.322,Y 20.6536,Z 60,A 65.8269,B 24.7918,C -3.3271,E1 25.045,E2 -703.4108} C_DIS
LIN {X 4.9273,Y 21.0307,Z 60,A 69.605,B 24.7915,C -3.3289,E1 25.0348,E2 -707.1874} C_DIS
LIN {X 3.7264,Y 21.2766,Z 60,A 73.1235,B 24.7911,C -3.3322,E1 25.0251,E2 -710.7097} C_DIS
LIN {X 2.256,Y 21.4819,Z 60,A 77.5184,B 24.7906,C -3.3362,E1 25.0129,E2 -715.111} C_DIS
LIN {X 0.0876,Y 21.5996,Z 60,A 82.7501,B 24.7911,C -3.332,E1 24.9984,E2 -720.3313} C_DIS
LIN {X -1.5438,Y 21.5445,Z 60,A 87.1243,B 24.7913,C -3.3308,E1 24.9862,E2 -724.7037} C_DIS
LIN {X -2.9369,Y 21.3998,Z 60,A 91.1442,B 24.7913,C -3.3306,E1 24.975,E2 -728.7261} C_DIS
LIN {X -4.6365,Y 21.0965,Z 60,A 95.5701,B 24.7919,C -3.326,E1 24.9629,E2 -733.146} C_DIS
LIN {X -5.7832,Y 20.8111,Z 60,A 98.709,B 24.7923,C -3.3229,E1 24.9545,E2 -736.2823} C_DIS
LIN {X -7.2973,Y 20.3299,Z 60,A 102.5222,B 24.7932,C -3.3156,E1 24.9444,E2 -740.0851} C_DIS
LIN {X -8.1851,Y 19.9891,Z 60,A 105.7744,B 24.7931,C -3.3164,E1 24.936,E2 -743.3466} C_DIS
LIN {X -9.7653,Y 19.2666,Z 60,A 109.5406,B 24.7945,C -3.3047,E1 24.9265,E2 -747.0944} C_DIS
LIN {X -10.7262,Y 18.7488,Z 60,A 112.9016,B 24.7948,C -3.3024,E1 24.9183,E2 -750.4595} C_DIS
LIN {X -11.7592,Y 18.1189,Z 60,A 116.3943,B 24.7954,C -3.298,E1 24.9101,E2 -753.9529} C_DIS
LIN {X -12.8212,Y 17.3835,Z 60,A 119.7916,B 24.7962,C -3.2911,E1 24.9024,E2 -757.3455} C_DIS
LIN {X -14.1496,Y 16.3206,Z 60,A 124.2945,B 24.7975,C -3.2813,E1 24.8928,E2 -761.8423} C_DIS
LIN {X -15.6693,Y 14.8677,Z 60,A 129.8744,B 24.7991,C -3.2683,E1 24.8818,E2 -767.4147} C_DIS
LIN {X -16.9347,Y 13.408,Z 60,A 135.0217,B 24.8006,C -3.2556,E1 24.8726,E2 -772.5551} C_DIS
LIN {X -17.8822,Y 12.1158,Z 60,A 139.2715,B 24.802,C -3.2443,E1 24.8658,E2 -776.7987} C_DIS
LIN {X -18.7036,Y 10.8021,Z 60,A 142.3228,B 24.804,C -3.2284,E1 24.8613,E2 -779.8276} C_DIS
LIN {X -19.2578,Y 9.7829,Z 60,A 146.61,B 24.8044,C -3.2248,E1 24.8557,E2 -784.1288} C_DIS
LIN {X -19.8954,Y 8.4092,Z 60,A 150.7981,B 24.8058,C -3.2137,E1 24.851,E2 -788.3136} C_DIS
LIN {X -20.5869,Y 6.5365,Z 60,A 155.4322,B 24.808,C -3.1951,E1 24.8468,E2 -792.9294} C_DIS
LIN {X -20.926,Y 5.353,Z 60,A 159.4723,B 24.8088,C -3.1883,E1 24.8439,E2 -796.9766} C_DIS
LIN {X -21.2985,Y 3.5975,Z 60,A 165.016,B 24.8102,C -3.1767,E1 24.8411,E2 -802.5255} C_DIS
LIN {X -21.5985,Y 0.1096,Z 60,A 173.2201,B 24.8142,C -3.1433,E1 24.8398,E2 -810.6989} C_DIS
LIN {X -21.5178,Y -1.8797,Z 60,A 178.9781,B 24.8159,C -3.1289,E1 24.8408,E2 -816.457} C_DIS
LIN {X -21.2997,Y -3.5901,Z 60,A -176.8642,B 24.8178,C -3.1133,E1 24.8425,E2 -820.602} C_DIS
LIN {X -21.0129,Y -5.0012,Z 60,A -173.0471,B 24.8191,C -3.1018,E1 24.8448,E2 -824.4141} C_DIS
LIN {X -20.5088,Y -6.7768,Z 60,A -167.1286,B 24.8203,C -3.092,E1 24.8497,E2 -830.3431} C_DIS
LIN {X -19.8356,Y -8.5495,Z 60,A -161.7444,B 24.8217,C -3.0796,E1 24.8555,E2 -835.7274} C_DIS
LIN {X -18.4096,Y -11.2985,Z 60,A -154.2911,B 24.8246,C -3.0546,E1 24.8657,E2 -843.1598} C_DIS
LIN {X -17.1165,Y -13.1749,Z 60,A -148.5877,B 24.8265,C -3.0384,E1 24.875,E2 -848.8524} C_DIS
LIN {X -16.1489,Y -14.3452,Z 60,A -144.631,B 24.8275,C -3.0291,E1 24.8822,E2 -852.8048} C_DIS
LIN {X -15.2948,Y -15.2514,Z 60,A -140.9291,B 24.8281,C -3.0244,E1 24.8894,E2 -856.5111} C_DIS
LIN {X -13.8614,Y -16.566,Z 60,A -135.3495,B 24.8289,C -3.0169,E1 24.9012,E2 -862.0949} C_DIS
LIN {X -11.6703,Y -18.1755,Z 60,A -128.6437,B 24.8306,C -3.0025,E1 24.9165,E2 -868.7891} C_DIS
LIN {X -10.1143,Y -19.0857,Z 60,A -124.3064,B 24.8316,C -2.9935,E1 24.927,E2 -873.1175} C_DIS
LIN {X -8.9381,Y -19.6634,Z 60,A -120.1242,B 24.8316,C -2.994,E1 24.9377,E2 -877.3113} C_DIS
LIN {X -7.2862,Y -20.3335,Z 60,A -116.1221,B 24.8325,C -2.9851,E1 24.948,E2 -881.3007} C_DIS
LIN {X -6.0602,Y -20.7323,Z 60,A -112.381,B 24.8325,C -2.9848,E1 24.958,E2 -885.0475} C_DIS
LIN {X -4.5679,Y -21.1113,Z 60,A -108.2186,B 24.8327,C -2.9833,E1 24.9694,E2 -889.2119} C_DIS
LIN {X -3.1957,Y -21.3625,Z 60,A -104.2909,B 24.8327,C -2.9839,E1 24.9802,E2 -893.1446} C_DIS
LIN {X -1.9381,Y -21.5128,Z 60,A -101.1634,B 24.8329,C -2.9819,E1 24.9889,E2 -896.2693} C_DIS
LIN {X -0.1005,Y -21.6,Z 60,A -96.4981,B 24.8329,C -2.981,E1 25.0019,E2 -900.9329} C_DIS
LIN {X -0.1005,Y -21.6,Z 60,A -96.4981,B 24.8329,C -2.981,E1 25.0019,E2 -900.9329} C_DIS
Enddeposition()
LIN {X 0.0251,Y -20.6414,Z 60,A -95.8983,B 24.8309,C -2.9993,E1 25.0037,E2 -901.5763} C_DIS
Startdeposition()
$VEL.CP = VEL_PRINT
LIN {X -0.664,Y -20.6313,Z 60,A -100.0073,B 24.8327,C -2.9836,E1 24.9921,E2 -897.4296} C_DIS
LIN {X -2.1215,Y -20.5326,Z 60,A -103.7702,B 24.8325,C -2.9857,E1 24.9817,E2 -893.6699} C_DIS
LIN {X -3.7242,Y -20.3034,Z 60,A -108.6445,B 24.8325,C -2.9845,E1 24.9682,E2 -888.7883} C_DIS
LIN {X -5.1194,Y -19.9968,Z 60,A -113.379,B 24.8329,C -2.9819,E1 24.9553,E2 -884.0409} C_DIS
LIN {X -7.7579,Y -19.1283,Z 60,A -121.0786,B 24.8321,C -2.9886,E1 24.9352,E2 -876.3418} C_DIS
LIN {X -10.1472,Y -17.976,Z 60,A -127.8154,B 24.8307,C -3.001,E1 24.9185,E2 -869.6163} C_DIS
LIN {X -12.1913,Y -16.6562,Z 60,A -135.0343,B 24.8298,C -3.0093,E1 24.9018,E2 -862.393} C_DIS
LIN {X -14.3253,Y -14.8601,Z 60,A -143.7198,B 24.8286,C -3.0199,E1 24.8839,E2 -853.698} C_DIS
LIN {X -16.8532,Y -11.9172,Z 60,A -154.0799,B 24.8255,C -3.0465,E1 24.866,E2 -843.3528} C_DIS
LIN {X -18.1806,Y -9.7746,Z 60,A -160.5848,B 24.8232,C -3.0666,E1 24.8569,E2 -836.8621} C_DIS
LIN {X -19.0521,Y -7.9436,Z 60,A -165.6553,B 24.8212,C -3.0842,E1 24.8512,E2 -831.806} C_DIS
LIN {X -19.6397,Y -6.3527,Z 60,A -170.6385,B 24.8197,C -3.0967,E1 24.8466,E2 -826.8244} C_DIS
LIN {X -20.1352,Y -4.5455,Z 60,A -176.221,B 24.8181,C -3.1108,E1 24.8428,E2 -821.243} C_DIS
LIN {X -20.4533,Y -2.7854,Z 60,A 179.4739,B 24.816,C -3.1282,E1 24.8409,E2 -816.954} C_DIS
LIN {X -20.5774,Y -1.6249,Z 60,A 176.1543,B 24.8149,C -3.1379,E1 24.8401,E2 -813.6377} C_DIS
LIN {X -20.6404,Y -0.1888,Z 60,A 172.5259,B 24.8132,C -3.1515,E1 24.8398,E2 -810.0202} C_DIS
LIN {X -20.6154,Y 1.0407,Z 60,A 167.7565,B 24.8125,C -3.1575,E1 24.8403,E2 -805.2363} C_DIS
LIN {X -20.3688,Y 3.3481,Z 60,A 162.3525,B 24.8097,C -3.1811,E1 24.8423,E2 -799.8567} C_DIS
LIN {X -20.1551,Y 4.4569,Z 60,A 158.7886,B 24.8087,C -3.1893,E1 24.8443,E2 -796.2913} C_DIS
LIN {X -19.7412,Y 6.0305,Z 60,A 154.6326,B 24.8069,C -3.2043,E1 24.8474,E2 -792.1473} C_DIS
LIN {X -19.3122,Y 7.288,Z 60,A 150.4555,B 24.8058,C -3.2136,E1 24.8514,E2 -787.9687} C_DIS
LIN {X -18.7761,Y 8.5758,Z 60,A 146.7968,B 24.8043,C -3.2257,E1 24.8555,E2 -784.3189} C_DIS
LIN {X -18.1325,Y 9.864,Z 60,A 142.6938,B 24.803,C -3.2367,E1 24.8608,E2 -780.2204} C_DIS
LIN {X -17.2962,Y 11.2664,Z 60,A 138.584,B 24.8012,C -3.2508,E1 24.8668,E2 -776.1233} C_DIS
LIN {X -16.4626,Y 12.4531,Z 60,A 134.2835,B 24.8001,C -3.2603,E1 24.8738,E2 -771.8247} C_DIS
LIN {X -15.8138,Y 13.2673,Z 60,A 131.0049,B 24.7994,C -3.266,E1 24.8796,E2 -768.5447} C_DIS
LIN {X -14.598,Y 14.5948,Z 60,A 125.8709,B 24.798,C -3.2773,E1 24.8896,E2 -763.4156} C_DIS
LIN {X -13.3646,Y 15.7296,Z 60,A 121.8815,B 24.7963,C -3.2905,E1 24.8978,E2 -759.4419} C_DIS
LIN {X -12.1914,Y 16.6572,Z 60,A 117.4076,B 24.7954,C -3.2975,E1 24.9078,E2 -754.9685} C_DIS
LIN {X -10.7995,Y 17.5914,Z 60,A 111.9317,B 24.7949,C -3.3022,E1 24.9207,E2 -749.4863} C_DIS
LIN {X -9.005,Y 18.5743,Z 60,A 106.6635,B 24.7935,C -3.3133,E1 24.9337,E2 -744.2302} C_DIS
LIN {X -7.2796,Y 19.3153,Z 60,A 101.7996,B 24.7924,C -3.3221,E1 24.9463,E2 -739.3766} C_DIS
LIN {X -5.5795,Y 19.8732,Z 60,A 96.6584,B 24.7918,C -3.3266,E1 24.96,E2 -734.2374} C_DIS
LIN {X -4.2751,Y 20.1943,Z 60,A 93.2781,B 24.7911,C -3.3319,E1 24.9692,E2 -730.8653} C_DIS
LIN {X -3.2306,Y 20.3878,Z 60,A 90.4208,B 24.7908,C -3.3346,E1 24.977,E2 -728.0114} C_DIS
LIN {X -1.9552,Y 20.5489,Z 60,A 85.8662,B 24.7913,C -3.3305,E1 24.9897,E2 -723.4444} C_DIS
LIN {X 0.7769,Y 20.6271,Z 60,A 78.2782,B 24.7911,C -3.3319,E1 25.0108,E2 -715.8602} C_DIS
LIN {X 2.4394,Y 20.497,Z 60,A 74.5558,B 24.7904,C -3.3375,E1 25.0211,E2 -712.1533} C_DIS
LIN {X 3.4645,Y 20.3493,Z 60,A 70.6729,B 24.7914,C -3.3296,E1 25.0319,E2 -708.2556} C_DIS
LIN {X 6.166,Y 19.6994,Z 60,A 62.9049,B 24.7921,C -3.3243,E1 25.0528,E2 -700.4877} C_DIS
LIN {X 7.8373,Y 19.0961,Z 60,A 57.2774,B 24.7933,C -3.3143,E1 25.0674,E2 -694.849} C_DIS
LIN {X 10.8569,Y 17.5564,Z 60,A 49.3023,B 24.7935,C -3.3131,E1 25.0868,E2 -686.8942} C_DIS
LIN {X 12.2205,Y 16.6356,Z 60,A 44.9298,B 24.7942,C -3.3073,E1 25.0968,E2 -682.523} C_DIS
LIN {X 13.5129,Y 15.6045,Z 60,A 40.0256,B 24.7956,C -3.2962,E1 25.1074,E2 -677.6112} C_DIS
LIN {X 14.7046,Y 14.4868,Z 60,A 35.7633,B 24.7965,C -3.2893,E1 25.1159,E2 -673.3505} C_DIS
LIN {X 15.4668,Y 13.67,Z 60,A 32.71,B 24.7972,C -3.283,E1 25.1216,E2 -670.2958} C_DIS
LIN {X 16.57,Y 12.3098,Z 60,A 27.5772,B 24.799,C -3.2692,E1 25.1304,E2 -665.1545} C_DIS
LIN {X 17.5494,Y 10.8682,Z 60,A 22.8007,B 24.8004,C -3.2577,E1 25.1377,E2 -660.3745} C_DIS
LIN {X 18.778,Y 8.5716,Z 60,A 14.641,B 24.8038,C -3.2296,E1 25.1479,E2 -652.1917} C_DIS
LIN {X 19.5794,Y 6.5362,Z 60,A 9.7607,B 24.8046,C -3.2235,E1 25.1525,E2 -647.3243} C_DIS
LIN {X 20.0223,Y 5.0183,Z 60,A 5.4294,B 24.8061,C -3.2111,E1 25.1557,E2 -642.9885} C_DIS
LIN {X 20.3459,Y 3.4848,Z 60,A 0.9279,B 24.8078,C -3.1965,E1 25.158,E2 -638.4787} C_DIS
LIN {X 20.5333,Y 2.1155,Z 60,A -2.9203,B 24.8093,C -3.1846,E1 25.1593,E2 -634.6251} C_DIS
LIN {X 20.6402,Y 0.2864,Z 60,A -7.688,B 24.8108,C -3.1719,E1 25.1598,E2 -629.8556} C_DIS
LIN {X 20.6293,Y -0.7264,Z 60,A -10.8065,B 24.8122,C -3.1602,E1 25.1595,E2 -626.7278} C_DIS
LIN {X 20.5256,Y -2.1877,Z 60,A -14.1729,B 24.8129,C -3.1543,E1 25.1587,E2 -623.3676} C_DIS
LIN {X 20.3671,Y -3.3584,Z 60,A -18.1784,B 24.815,C -3.137,E1 25.157,E2 -619.3445} C_DIS
LIN {X 20.0339,Y -4.9692,Z 60,A -22.0062,B 24.8158,C -3.1301,E1 25.1547,E2 -615.5227} C_DIS
LIN {X 19.7249,Y -6.0836,Z 60,A -25.6737,B 24.8175,C -3.1159,E1 25.1518,E2 -611.8424} C_DIS
LIN {X 19.0308,Y -7.9945,Z 60,A -31.5494,B 24.8197,C -3.0968,E1 25.1458,E2 -605.954} C_DIS
LIN {X 18.162,Y -9.81,Z 60,A -36.8338,B 24.8212,C -3.0836,E1 25.1391,E2 -600.6665} C_DIS
LIN {X 17.3606,Y -11.1671,Z 60,A -41.0064,B 24.8224,C -3.0734,E1 25.133,E2 -596.4909} C_DIS
LIN {X 16.5831,Y -12.2913,Z 60,A -44.5191,B 24.8233,C -3.0659,E1 25.1273,E2 -592.9776} C_DIS
LIN {X 15.8853,Y -13.1815,Z 60,A -47.5005,B 24.8241,C -3.0593,E1 25.1221,E2 -589.9944} C_DIS
LIN {X 14.986,Y -14.1957,Z 60,A -51.4621,B 24.8253,C -3.0482,E1 25.1147,E2 -586.0241} C_DIS
LIN {X 14.1966,Y -14.9852,Z 60,A -54.887,B 24.8265,C -3.0381,E1 25.1078,E2 -582.5893} C_DIS
LIN {X 13.0033,Y -16.0313,Z 60,A -58.7598,B 24.8271,C -3.0332,E1 25.0996,E2 -578.72} C_DIS
LIN {X 11.6834,Y -17.0175,Z 60,A -63.7147,B 24.8285,C -3.0206,E1 25.0883,E2 -573.7527} C_DIS
LIN {X 10.6547,Y -17.6798,Z 60,A -67.1952,B 24.8293,C -3.0137,E1 25.0801,E2 -570.2668} C_DIS
LIN {X 9.2246,Y -18.4661,Z 60,A -71.365,B 24.8298,C -3.0092,E1 25.0698,E2 -566.0981} C_DIS
LIN {X 8.0751,Y -18.9968,Z 60,A -75.6451,B 24.8311,C -2.9978,E1 25.0588,E2 -561.8013} C_DIS
LIN {X 6.1947,Y -19.6903,Z 60,A -80.9421,B 24.8316,C -2.9931,E1 25.0448,E2 -556.5036} C_DIS
LIN {X 3.9181,Y -20.2666,Z 60,A -88.2271,B 24.8329,C -2.9815,E1 25.0249,E2 -549.2007} C_DIS
LIN {X 2.0465,Y -20.5404,Z 60,A -93.0653,B 24.8329,C -2.9815,E1 25.0115,E2 -544.3659} C_DIS
LIN {X 0.0251,Y -20.6414,Z 60,A -95.8983,B 24.8309,C -2.9993,E1 25.0037,E2 -541.5763} C_DIS
Enddeposition()
LIN {X 0.0251,Y -20.6414,Z 60,A -95.8983,B 24.8309,C -2.9993,E1 25.0037,E2 -541.5763} C_DIS
Startdeposition()
$VEL.CP = VEL_PRINT
LIN {X 1.0666,Y -19.6546,Z 60,A -92.8753,B 24.829,C -3.0166,E1 25.0122,E2 -544.6394} C_DIS
LIN {X 2.7256,Y -19.4943,Z 60,A -87.7917,B 24.8284,C -3.0212,E1 25.0264,E2 -549.7301} C_DIS
LIN {X 4.5714,Y -19.1454,Z 60,A -82.8171,B 24.8284,C -3.0222,E1 25.0399,E2 -554.7008} C_DIS
LIN {X 6.11,Y -18.7114,Z 60,A -77.8682,B 24.8275,C -3.0297,E1 25.0532,E2 -559.6588} C_DIS
LIN {X 7.6929,Y -18.1183,Z 60,A -73.5531,B 24.8273,C -3.0315,E1 25.0644,E2 -563.9686} C_DIS
LIN {X 8.7874,Y -17.6116,Z 60,A -69.9845,B 24.8266,C -3.0375,E1 25.0734,E2 -567.542} C_DIS
LIN {X 9.8341,Y -17.0512,Z 60,A -65.8976,B 24.8253,C -3.0486,E1 25.0834,E2 -571.6434} C_DIS
LIN {X 11.6051,Y -15.899,Z 60,A -59.5343,B 24.8237,C -3.0625,E1 25.098,E2 -578.0179} C_DIS
LIN {X 13.3771,Y -14.44,Z 60,A -53.6929,B 24.8229,C -3.0697,E1 25.1104,E2 -583.8537} C_DIS
LIN {X 14.5425,Y -13.2654,Z 60,A -48.249,B 24.8208,C -3.087,E1 25.1209,E2 -589.315} C_DIS
LIN {X 15.5063,Y -12.1252,Z 60,A -44.6043,B 24.8203,C -3.0917,E1 25.1273,E2 -592.9539} C_DIS
LIN {X 16.1722,Y -11.2213,Z 60,A -40.7778,B 24.8187,C -3.1056,E1 25.1335,E2 -596.7948} C_DIS
LIN {X 17.3724,Y -9.2541,Z 60,A -33.9269,B 24.8163,C -3.1258,E1 25.1431,E2 -603.6581} C_DIS
LIN {X 18.1103,Y -7.7098,Z 60,A -28.9675,B 24.8146,C -3.1402,E1 25.1487,E2 -608.6246} C_DIS
LIN {X 18.7686,Y -5.9313,Z 60,A -23.7886,B 24.813,C -3.1536,E1 25.1534,E2 -613.806} C_DIS
LIN {X 19.2556,Y -4.0831,Z 60,A -18.0111,B 24.8107,C -3.1728,E1 25.1571,E2 -619.5956} C_DIS
LIN {X 19.5353,Y -2.4132,Z 60,A -14.0047,B 24.8099,C -3.1791,E1 25.1588,E2 -623.5935} C_DIS
LIN {X 19.6296,Y -1.456,Z 60,A -11.0289,B 24.8087,C -3.1896,E1 25.1595,E2 -626.5764} C_DIS
LIN {X 19.6822,Y -0.1798,Z 60,A -6.9848,B 24.8069,C -3.2044,E1 25.1598,E2 -630.6315} C_DIS
Enddeposition()
END
